(* IEC 61131-3 sources: Elmo_Master/test/Reports_Lasal/C78_20260806_preemption_cleanup_split (part 2) *)

	resourceBusy := FALSE;
	case ResourceKind of
		LMC_OWNER_RESOURCE_LMC_HOME_ENGINE:
			resourceBusy := (OwnershipState[7]$UDINT <> 0) |
				(OwnershipState[8]$UDINT <> 0) |
				(OwnershipState[9]$UDINT <> 0);
		LMC_OWNER_RESOURCE_DS402_HOME_ENGINE:
			resourceBusy := (OwnershipState[10]$UDINT <> 0) |
				(OwnershipState[11]$UDINT <> 0) |
				(OwnershipState[12]$UDINT <> 0);
		LMC_OWNER_RESOURCE_DIAGNOSTICS_SDO_ENGINE:
			resourceBusy := (OwnershipState[13]$UDINT <> 0) |
				(OwnershipState[14]$UDINT <> 0) |
				(OwnershipState[15]$UDINT <> 0);
	else
	end_case;
	if resourceBusy then
		Result := -2;
		RETURN;
	end_if;

	groupLeaseTransition :=
		(OwnerKind = LMC_OWNER_KIND_GROUP) &
		((CommandId = 0x20A4) | (CommandId = 0x7D22) |
		 (CommandId = 0x2048));
	groupStopTransition :=
		(OwnerKind = LMC_OWNER_KIND_GROUP) & (CommandId = 0x2085);

	// A direct safety command against a Group member protects the complete
	// exact lease mask. Unknown Group state widens to the administrative mask
	// and is forced to quarantine after the physical safety observation.
	if (OwnerKind = LMC_OWNER_KIND_DIRECT) & safetyPreemption &
	   (referenceAxisMask <> 0) then
		axisIndex := TO_DINT(Reference);
		recordBase := LMC_OWNER_GLOBAL_SLOTS +
			((axisIndex - 1) * LMC_OWNER_AXIS_STRIDE);
		if (OwnershipState[recordBase + 1] = LMC_OWNER_STATE_GROUP_LEASE) |
		   (OwnershipState[recordBase + 1] = LMC_OWNER_STATE_GROUP_ACTIVE) then
			if (OwnershipState[recordBase + 11]$UDINT <> 0) &
			   (OwnershipState[recordBase + 11]$UDINT <=
			    LMC_OWNER_ROBOT_AXIS_MASK) then
				effectiveAxisMask :=
					OwnershipState[recordBase + 11]$UDINT;
			else
				effectiveAxisMask := LMC_OWNER_ROBOT_AXIS_MASK;
			end_if;
			forceQuarantine := TRUE;
		end_if;
	end_if;

	if groupStopTransition then
		recordBase := LMC_OWNER_GLOBAL_SLOTS;
		if ((OwnershipState[recordBase + 1] = LMC_OWNER_STATE_GROUP_LEASE) |
		    (OwnershipState[recordBase + 1] = LMC_OWNER_STATE_GROUP_ACTIVE)) &
		   (OwnershipState[recordBase + 2] = LMC_OWNER_KIND_GROUP) &
		   (OwnershipState[recordBase + 11]$UDINT =
		    LMC_OWNER_PROFILE_AXIS_MASK) then
			effectiveAxisMask := LMC_OWNER_PROFILE_AXIS_MASK;
		else
			effectiveAxisMask := LMC_OWNER_ROBOT_AXIS_MASK;
			forceQuarantine := TRUE;
		end_if;
	end_if;

	// Repeated safety commands reuse the immutable live lineage. Admission
	// returns +1 for a no-native ACK and +2 for one monotonic PowerOff call.
	repeatCandidate := safetyPreemption &
		((CommandId = LMC_OWNER_COMMAND_AXIS_STOP) |
		 (CommandId = LMC_OWNER_COMMAND_AXIS_POWER) |
		 (CommandId = LMC_OWNER_COMMAND_GROUP_DISABLE) |
		 (CommandId = LMC_OWNER_COMMAND_GROUP_STOP) |
		 (CommandId = LMC_OWNER_COMMAND_GROUP_POWER_OFF));
	if repeatCandidate then
		if OwnerKind = LMC_OWNER_KIND_DIRECT then
			if (Reference >= 1) & (Reference <= LMC_OWNER_AXIS_COUNT) then
			repeatRecordBase := LMC_OWNER_GLOBAL_SLOTS +
				((TO_DINT(Reference) - 1) * LMC_OWNER_AXIS_STRIDE);
			if (OwnershipState[repeatRecordBase + 2] =
			    LMC_OWNER_KIND_DIRECT) &
			   (OwnershipState[repeatRecordBase + 13] =
			    LMC_OWNER_RESOURCE_AXIS) &
			   (OwnershipState[repeatRecordBase + 14] =
			    LMC_OWNER_ADMISSION_SAFETY) then
				repeatFound := TRUE;
			end_if;
			end_if;
		else
			axisIndex := 1;
			while axisIndex <= LMC_OWNER_AXIS_COUNT do
				recordBase := LMC_OWNER_GLOBAL_SLOTS +
					((axisIndex - 1) * LMC_OWNER_AXIS_STRIDE);
				if (OwnershipState[recordBase + 2] =
				    LMC_OWNER_KIND_GROUP) &
				   (OwnershipState[recordBase + 13] =
				    LMC_OWNER_RESOURCE_AXIS) &
				   (OwnershipState[recordBase + 14] =
				    LMC_OWNER_ADMISSION_SAFETY) then
					if repeatFound = FALSE then
						repeatRecordBase := recordBase;
						repeatFound := TRUE;
					elsif (OwnershipState[repeatRecordBase + 4] <>
					       OwnershipState[recordBase + 4]) |
					      (OwnershipState[repeatRecordBase + 5] <>
					       OwnershipState[recordBase + 5]) then
						OwnershipState[24] := 1;
						Result := -3;
						RETURN;
					end_if;
				end_if;
				axisIndex += 1;
			end_while;
		end_if;
	end_if;
	if repeatFound then
		repeatState := OwnershipState[repeatRecordBase + 1];
		if repeatState = LMC_OWNER_STATE_QUARANTINED then
			OwnershipState[24] := 1;
			Result := -3;
			RETURN;
		end_if;
		repeatValid := (repeatState = LMC_OWNER_STATE_RESERVED) |
			(repeatState = LMC_OWNER_STATE_SAFETY_PREEMPTING);
		repeatCommand := OwnershipState[repeatRecordBase + 3];
		repeatReference := OwnershipState[repeatRecordBase + 12];
		repeatOwnerKind := OwnershipState[repeatRecordBase + 2];
		repeatAxisMask := OwnershipState[repeatRecordBase + 11]$UDINT;
		repeatAdmissionToken :=
			OwnershipState[repeatRecordBase + 4]$UDINT;
		repeatOwnerGeneration :=
			OwnershipState[repeatRecordBase + 5]$UDINT;
		repeatSession := OwnershipState[repeatRecordBase + 6]$UDINT;
		repeatSequence := OwnershipState[repeatRecordBase + 7]$UDINT;
		repeatIdentitySize := OwnershipState[repeatRecordBase + 15]$UDINT;
		repeatValid := repeatValid &
			(repeatAxisMask <> 0) &
			(repeatAxisMask <= LMC_OWNER_ROBOT_AXIS_MASK) &
			(repeatAdmissionToken <> 0) &
			(repeatOwnerGeneration <> 0) &
			(repeatSession <> 0) & (repeatSequence <> 0) &
			(((repeatOwnerKind = LMC_OWNER_KIND_DIRECT) &
			  (repeatReference = TO_DINT(Reference)) &
			  ((repeatCommand = LMC_OWNER_COMMAND_AXIS_STOP) |
			   (repeatCommand = LMC_OWNER_COMMAND_AXIS_POWER))) |
			 ((repeatOwnerKind = LMC_OWNER_KIND_GROUP) &
			  (repeatReference = 0x0100) &
			  ((repeatCommand = LMC_OWNER_COMMAND_GROUP_DISABLE) |
			   (repeatCommand = LMC_OWNER_COMMAND_GROUP_STOP) |
			   (repeatCommand = LMC_OWNER_COMMAND_GROUP_POWER_OFF))));
		if repeatValid then
			if repeatState = LMC_OWNER_STATE_RESERVED then
				repeatValidationResult := ValidateAxisOwnershipIdentity(
					CommandId:=repeatCommand$UINT,
					Reference:=repeatReference$UINT,
					ExpectedAxisMask:=repeatAxisMask,
					OwnerKind:=repeatOwnerKind$UINT,
					ResourceKind:=LMC_OWNER_RESOURCE_AXIS,
					AdmissionMode:=LMC_OWNER_ADMISSION_SAFETY,
					CallerSessionEpoch:=repeatSession,
					RequestSequence:=repeatSequence,
					AdmissionToken:=repeatAdmissionToken,
					OwnerGeneration:=repeatOwnerGeneration,
					RequiredPhase:=LMC_OWNER_PHASE_RESERVED,
					pIdentity:=(#OwnershipState[repeatRecordBase + 16])$^void,
					IdentitySize:=repeatIdentitySize);
			else
				repeatValidationResult := ValidateAxisOwnershipIdentity(
				CommandId:=repeatCommand$UINT,
				Reference:=repeatReference$UINT,
				ExpectedAxisMask:=repeatAxisMask,
				OwnerKind:=repeatOwnerKind$UINT,
				ResourceKind:=LMC_OWNER_RESOURCE_AXIS,
				AdmissionMode:=LMC_OWNER_ADMISSION_SAFETY,
				CallerSessionEpoch:=repeatSession,
				RequestSequence:=repeatSequence,
				AdmissionToken:=repeatAdmissionToken,
				OwnerGeneration:=repeatOwnerGeneration,
				RequiredPhase:=LMC_OWNER_PHASE_ACTIVE,
				pIdentity:=(#OwnershipState[repeatRecordBase + 16])$^void,
				IdentitySize:=repeatIdentitySize);
			end_if;
			repeatValid := repeatValidationResult = 0;
		end_if;
		if repeatState = LMC_OWNER_STATE_RESERVED then
			if repeatValid then
				Result := -2;
			else
				OwnershipState[24] := 1;
				Result := -3;
			end_if;
			RETURN;
		end_if;
		if repeatValid then
			axisIndex := 1;
			while axisIndex <= LMC_OWNER_AXIS_COUNT do
				case axisIndex of
					1: axisBit := 0x00000001;
					2: axisBit := 0x00000002;
					3: axisBit := 0x00000004;
					4: axisBit := 0x00000008;
					5: axisBit := 0x00000010;
					6: axisBit := 0x00000020;
					7: axisBit := 0x00000040;
					8: axisBit := 0x00000080;
					9: axisBit := 0x00000100;
				else
					axisBit := 0;
				end_case;
				if (repeatAxisMask and axisBit) <> 0 then
					observerBase := (axisIndex - 1) *
						LMC_OWNER_OBSERVER_STRIDE;
					observerFlags :=
						OwnershipObserverState[observerBase + 5]$UDINT;
					if (OwnershipObserverState[observerBase]$UDINT <>
					    (LMC_OWNER_OBSERVER_MAGIC + TO_UDINT(axisIndex))) |
					   (OwnershipObserverState[observerBase + 1]$UDINT <>
					    repeatAdmissionToken) |
					   (OwnershipObserverState[observerBase + 2]$UDINT <>
					    repeatOwnerGeneration) |
					   ((observerFlags and
					     (0xFFFFFFFF xor LMC_OWNER_OBSERVER_KNOWN_MASK)) <> 0) then
						repeatValid := FALSE;
					end_if;
					if (observerFlags and
					    LMC_OWNER_OBSERVER_PREEMPTED) <> 0 then
						repeatPreemptedSeen := TRUE;
						if (OwnershipObserverState[observerBase + 9] = 0) |
						   (OwnershipObserverState[observerBase + 10] = 0) |
						   (OwnershipObserverState[observerBase + 11] = 0) then
							repeatValid := FALSE;
						end_if;
					elsif (OwnershipObserverState[observerBase + 9] <> 0) |
					      (OwnershipObserverState[observerBase + 10] <> 0) |
					      (OwnershipObserverState[observerBase + 11] <> 0) then
						repeatValid := FALSE;
					end_if;
					if repeatRecordBase = (LMC_OWNER_GLOBAL_SLOTS +
					   ((axisIndex - 1) * LMC_OWNER_AXIS_STRIDE)) then
						repeatEscalated := (observerFlags and
							LMC_OWNER_OBSERVER_POWER_OFF_ESCALATED) <> 0;
						repeatForceQuarantine := (observerFlags and
							LMC_OWNER_OBSERVER_FORCE_QUARANTINE) <> 0;
					else
						if repeatEscalated <>
						   ((observerFlags and
						     LMC_OWNER_OBSERVER_POWER_OFF_ESCALATED) <> 0) then
							repeatValid := FALSE;
						end_if;
						if repeatForceQuarantine <>
						   ((observerFlags and
						     LMC_OWNER_OBSERVER_FORCE_QUARANTINE) <> 0) then
							repeatValid := FALSE;
						end_if;
					end_if;
				end_if;
				axisIndex += 1;
			end_while;
		end_if;
		if repeatValid & (repeatOwnerKind = LMC_OWNER_KIND_DIRECT) then
			if ((repeatAxisMask and referenceAxisMask) <> referenceAxisMask) |
			   ((repeatAxisMask <> referenceAxisMask) &
			    (repeatForceQuarantine = FALSE)) then
				repeatValid := FALSE;
			end_if;
		elsif repeatValid & (repeatOwnerKind = LMC_OWNER_KIND_GROUP) then
			if ((repeatCommand = LMC_OWNER_COMMAND_GROUP_DISABLE) &
			    (repeatAxisMask <> LMC_OWNER_PROFILE_AXIS_MASK)) |
			   ((repeatCommand = LMC_OWNER_COMMAND_GROUP_STOP) &
			    (repeatAxisMask <> LMC_OWNER_PROFILE_AXIS_MASK) &
			    (repeatAxisMask <> LMC_OWNER_ROBOT_AXIS_MASK)) |
			   ((repeatCommand = LMC_OWNER_COMMAND_GROUP_POWER_OFF) &
			    (repeatAxisMask <> LMC_OWNER_ROBOT_AXIS_MASK)) then
				repeatValid := FALSE;
			end_if;
		end_if;
		if repeatValid & repeatEscalated &
		   ((repeatCommand = LMC_OWNER_COMMAND_AXIS_POWER) |
		    (repeatCommand = LMC_OWNER_COMMAND_GROUP_POWER_OFF)) then
			repeatValid := FALSE;
		end_if;
		if repeatValid & repeatRootPresent then
			repeatRootForce :=
				(OwnershipPreemptedIdentityState[
				 LMC_OWNER_PREEMPT_HEADER_BASE + 1]$UDINT and
				 LMC_OWNER_PREEMPT_FLAG_FORCE_QUARANTINE) <> 0;
			if ((OwnershipPreemptedIdentityState[
			     LMC_OWNER_PREEMPT_HEADER_BASE + 1]$UDINT and
			     0x0000FFFF) <> LMC_OWNER_IDENTITY_VERSION) |
			   ((OwnershipPreemptedIdentityState[
			     LMC_OWNER_PREEMPT_HEADER_BASE + 1]$UDINT and
			     0xFFFE0000) <> 0) |
			   (repeatPreemptedSeen = FALSE) then
				repeatValid := FALSE;
			end_if;
			if repeatValid &
			   (repeatRootForce <> repeatForceQuarantine) then
				if repeatRootForce |
				   (repeatForceQuarantine = FALSE) |
				   (repeatEscalated = FALSE) |
				   (repeatOwnerKind <> LMC_OWNER_KIND_GROUP) |
				   (repeatAxisMask <> LMC_OWNER_PROFILE_AXIS_MASK) |
				   ((repeatCommand <> LMC_OWNER_COMMAND_GROUP_DISABLE) &
				    (repeatCommand <> LMC_OWNER_COMMAND_GROUP_STOP)) then
					repeatValid := FALSE;
				end_if;
			end_if;
			axisIndex := 1;
			while axisIndex <= LMC_OWNER_AXIS_COUNT do
				probeRecordBase :=
					(axisIndex - 1) * LMC_OWNER_AXIS_STRIDE;
				if (repeatPreemptedToken = 0) &
				   (OwnershipPreemptedState[probeRecordBase + 1] <>
				    LMC_OWNER_STATE_IDLE) &
				   ((OwnershipPreemptedState[probeRecordBase + 11]$UDINT and
				     repeatAxisMask) <> 0) then
					repeatPreemptedToken := OwnershipPreemptedState[
						probeRecordBase + 4]$UDINT;
					repeatPreemptedGeneration := OwnershipPreemptedState[
						probeRecordBase + 5]$UDINT;
				end_if;
				axisIndex += 1;
			end_while;
			if (repeatPreemptedToken = 0) |
			   (repeatPreemptedGeneration = 0) then
				repeatValid := FALSE;
			end_if;
		elsif repeatValid & repeatPreemptedSeen then
			repeatValid := FALSE;
		end_if;
		if repeatValid then
			if repeatEscalated &
			   (repeatCommand = LMC_OWNER_COMMAND_AXIS_STOP) &
			   ((CommandId = LMC_OWNER_COMMAND_AXIS_STOP) |
			    (CommandId = LMC_OWNER_COMMAND_AXIS_POWER)) then
				repeatMode := 1;
			elsif repeatEscalated &
			      ((repeatCommand = LMC_OWNER_COMMAND_GROUP_STOP) |
			       (repeatCommand = LMC_OWNER_COMMAND_GROUP_DISABLE)) &
			      ((CommandId = LMC_OWNER_COMMAND_GROUP_STOP) |
			       (CommandId = LMC_OWNER_COMMAND_GROUP_DISABLE) |
			       (CommandId = LMC_OWNER_COMMAND_GROUP_POWER_OFF)) then
				repeatMode := 1;
			elsif repeatCommand = TO_DINT(CommandId) then
				if (repeatCommand = LMC_OWNER_COMMAND_AXIS_STOP) |
				   (repeatCommand = LMC_OWNER_COMMAND_GROUP_STOP) then
					identityCompareResult := _memcmp(
						ptr1:=pIdentity,
						ptr2:=#OwnershipState[repeatRecordBase + 16],
						cntr:=repeatIdentitySize);
					if identityCompareResult = 0 then
						repeatMode := 1;
					end_if;
				else
					repeatMode := 1;
				end_if;
			elsif (repeatCommand = LMC_OWNER_COMMAND_AXIS_POWER) &
			      (CommandId = LMC_OWNER_COMMAND_AXIS_STOP) then
				repeatMode := 1;
			elsif (repeatCommand = LMC_OWNER_COMMAND_GROUP_POWER_OFF) &
			      ((CommandId = LMC_OWNER_COMMAND_GROUP_STOP) |
			       (CommandId = LMC_OWNER_COMMAND_GROUP_DISABLE)) then
				repeatMode := 1;
			elsif (repeatCommand = LMC_OWNER_COMMAND_AXIS_STOP) &
			      (CommandId = LMC_OWNER_COMMAND_AXIS_POWER) then
				if repeatEscalated then
					repeatMode := 1;
				else
					repeatMode := 2;
				end_if;
			elsif ((repeatCommand = LMC_OWNER_COMMAND_GROUP_STOP) |
			       (repeatCommand = LMC_OWNER_COMMAND_GROUP_DISABLE)) &
			      (CommandId = LMC_OWNER_COMMAND_GROUP_POWER_OFF) then
				if repeatEscalated then
					repeatMode := 1;
				else
					repeatMode := 2;
				end_if;
			end_if;
		end_if;
		if repeatValid = FALSE then
			OwnershipState[24] := 1;
			Result := -3;
			RETURN;
		end_if;
	end_if;
	if repeatRootPresent & safetyPreemption & (repeatMode = 0) then
		Result := -2;
		RETURN;
	end_if;

	if repeatMode = 0 then
	axisIndex := 1;
	while axisIndex <= LMC_OWNER_AXIS_COUNT do
		case axisIndex of
			1: axisBit := 0x00000001;
			2: axisBit := 0x00000002;
			3: axisBit := 0x00000004;
			4: axisBit := 0x00000008;
			5: axisBit := 0x00000010;
			6: axisBit := 0x00000020;
			7: axisBit := 0x00000040;
			8: axisBit := 0x00000080;
			9: axisBit := 0x00000100;
		else
			axisBit := 0;
		end_case;
		if (effectiveAxisMask and axisBit) <> 0 then
			recordBase := LMC_OWNER_GLOBAL_SLOTS +
				((axisIndex - 1) * LMC_OWNER_AXIS_STRIDE);
			if (OwnershipState[recordBase] <> axisIndex) |
			   (OwnershipState[recordBase + 35]$UDINT <>
			    (LMC_OWNER_AXIS_RECORD_MAGIC + TO_UDINT(axisIndex))) then
				Result := -3;
				RETURN;
			end_if;
			existingState := OwnershipState[recordBase + 1];
			existingOwnerKind := OwnershipState[recordBase + 2];
			if (existingState = LMC_OWNER_STATE_IDLE) &
			   ((OwnershipState[recordBase + 2] <> 0) |
			    (OwnershipState[recordBase + 3] <> 0) |
			    (OwnershipState[recordBase + 4] <> 0) |
			    (OwnershipState[recordBase + 5] <> 0) |
			    (OwnershipState[recordBase + 6] <> 0) |
			    (OwnershipState[recordBase + 7] <> 0) |
			    (OwnershipState[recordBase + 11] <> 0) |
			    (OwnershipState[recordBase + 13] <> 0) |
			    (OwnershipState[recordBase + 14] <> 0) |
			    (OwnershipState[recordBase + 15] <> 0)) then
				Result := -3;
				RETURN;
			end_if;
			if safetyPreemption &
			   (existingState = LMC_OWNER_STATE_SAFETY_PREEMPTING) then
				Result := -2;
				RETURN;
			end_if;

			// Validate the complete current identity header before it can be
			// copied to a lease or preemption bank.
			existingIdentityValid := existingState = LMC_OWNER_STATE_IDLE;
			if existingState <> LMC_OWNER_STATE_IDLE then
				if (OwnershipState[recordBase + 15] < 0) |
				   (OwnershipState[recordBase + 15]$UDINT > 1320) then
					Result := -3;
					RETURN;
				end_if;
				if existingOwnerKind = LMC_OWNER_KIND_GROUP then
					identityHeaderBase := LMC_OWNER_IDENTITY_GROUP_HEADER_BASE;
					existingIdentityValid :=
						(OwnershipIdentityState[identityHeaderBase]$UDINT =
						 LMC_OWNER_IDENTITY_GROUP_MAGIC) &
						(OwnershipIdentityState[identityHeaderBase + 1] =
						 LMC_OWNER_IDENTITY_VERSION) &
						(OwnershipIdentityState[identityHeaderBase + 2]$UDINT =
						 OwnershipState[recordBase + 15]$UDINT) &
						(OwnershipIdentityState[identityHeaderBase + 3]$UDINT =
						 OwnershipState[recordBase + 4]$UDINT) &
						(OwnershipIdentityState[identityHeaderBase + 4]$UDINT =
						 OwnershipState[recordBase + 5]$UDINT) &
						(OwnershipIdentityState[identityHeaderBase + 5]$UDINT =
						 OwnershipState[recordBase + 11]$UDINT) &
						(OwnershipIdentityState[identityHeaderBase + 6]$UDINT =
						 OwnershipState[recordBase + 6]$UDINT) &
						(OwnershipIdentityState[identityHeaderBase + 7]$UDINT =
						 OwnershipState[recordBase + 7]$UDINT) &
						(OwnershipIdentityState[identityHeaderBase + 8]$UDINT =
						 (TO_UDINT(OwnershipState[recordBase + 3]) or
						  (TO_UDINT(OwnershipState[recordBase + 12]) shl 16))) &
						(OwnershipIdentityState[identityHeaderBase + 9]$UDINT =
						 (TO_UDINT(OwnershipState[recordBase + 2]) or
						  (TO_UDINT(OwnershipState[recordBase + 13]) shl 8) or
						  (TO_UDINT(OwnershipState[recordBase + 14]) shl 16)));
				else
					identityHeaderBase := LMC_OWNER_IDENTITY_AXIS_HEADER_BASE +
						((axisIndex - 1) *
						 LMC_OWNER_IDENTITY_AXIS_HEADER_STRIDE);
					identityTailSize := 0;
					if OwnershipState[recordBase + 15]$UDINT >
					   LMC_OWNER_IDENTITY_PREFIX_BYTES then
						identityTailSize :=
							OwnershipState[recordBase + 15]$UDINT -
							LMC_OWNER_IDENTITY_PREFIX_BYTES;
					end_if;
					if (OwnershipState[recordBase + 12] < 1) |
					   (OwnershipState[recordBase + 12] >
					    LMC_OWNER_AXIS_COUNT) |
					   (identityTailSize > 8) then
						Result := -3;
						RETURN;
					end_if;
					identityTailOffset :=
						TO_UDINT(OwnershipState[recordBase + 12] - 1) * 8;
					existingIdentityValid :=
						(OwnershipIdentityState[identityHeaderBase]$UDINT =
						 (LMC_OWNER_IDENTITY_AXIS_MAGIC + TO_UDINT(axisIndex))) &
						(OwnershipIdentityState[identityHeaderBase + 1] =
						 LMC_OWNER_IDENTITY_VERSION) &
						(OwnershipIdentityState[identityHeaderBase + 2]$UDINT =
						 OwnershipState[recordBase + 15]$UDINT) &
						(OwnershipIdentityState[identityHeaderBase + 3]$UDINT =
						 OwnershipState[recordBase + 4]$UDINT) &
						(OwnershipIdentityState[identityHeaderBase + 4]$UDINT =
						 OwnershipState[recordBase + 5]$UDINT) &
						(OwnershipIdentityState[identityHeaderBase + 5]$UDINT =
						 OwnershipState[recordBase + 11]$UDINT) &
						(OwnershipIdentityState[identityHeaderBase + 6]$UDINT =
						 OwnershipState[recordBase + 6]$UDINT) &
						(OwnershipIdentityState[identityHeaderBase + 7]$UDINT =
						 OwnershipState[recordBase + 7]$UDINT) &
						(OwnershipIdentityState[identityHeaderBase + 8]$UDINT =
						 (TO_UDINT(OwnershipState[recordBase + 3]) or
						  (TO_UDINT(OwnershipState[recordBase + 12]) shl 16))) &
						(OwnershipIdentityState[identityHeaderBase + 9]$UDINT =
						 (TO_UDINT(OwnershipState[recordBase + 2]) or
						  (TO_UDINT(OwnershipState[recordBase + 13]) shl 8) or
						  (TO_UDINT(OwnershipState[recordBase + 14]) shl 16))) &
						(OwnershipIdentityState[identityHeaderBase + 10]$UDINT =
						 identityTailOffset) &
						(OwnershipIdentityState[identityHeaderBase + 11]$UDINT =
						 identityTailSize);
				end_if;
				if existingIdentityValid = FALSE then
					Result := -3;
					RETURN;
				end_if;
				// Every member of one captured tuple was created from one request.
				// Prove complete membership and byte-exact prefix coherence before
				// any backup publication or live ownership mutation.
				existingIdentityPrefixSize :=
					OwnershipState[recordBase + 15]$UDINT;
				if existingIdentityPrefixSize >
				   LMC_OWNER_IDENTITY_PREFIX_BYTES then
					existingIdentityPrefixSize :=
						LMC_OWNER_IDENTITY_PREFIX_BYTES;
				end_if;
				if (OwnershipState[recordBase + 4]$UDINT = 0) |
				   (OwnershipState[recordBase + 5]$UDINT = 0) |
				   (OwnershipState[recordBase + 6]$UDINT = 0) |
				   (OwnershipState[recordBase + 7]$UDINT = 0) |
				   (OwnershipState[recordBase + 11]$UDINT = 0) |
				   (OwnershipState[recordBase + 11]$UDINT >
				    LMC_OWNER_ROBOT_AXIS_MASK) |
				   ((OwnershipState[recordBase + 11]$UDINT and axisBit) = 0) then
					Result := -3;
					RETURN;
				end_if;
				probeAxisIndex := 1;
				while probeAxisIndex <= LMC_OWNER_AXIS_COUNT do
					case probeAxisIndex of
						1: probeAxisBit := 0x00000001;
						2: probeAxisBit := 0x00000002;
						3: probeAxisBit := 0x00000004;
						4: probeAxisBit := 0x00000008;
						5: probeAxisBit := 0x00000010;
						6: probeAxisBit := 0x00000020;
						7: probeAxisBit := 0x00000040;
						8: probeAxisBit := 0x00000080;
						9: probeAxisBit := 0x00000100;
					else
						probeAxisBit := 0;
					end_case;
					probeRecordBase := LMC_OWNER_GLOBAL_SLOTS +
						((probeAxisIndex - 1) * LMC_OWNER_AXIS_STRIDE);
					if (OwnershipState[recordBase + 11]$UDINT and
					    probeAxisBit) <> 0 then
						if (OwnershipState[probeRecordBase] <>
						    probeAxisIndex) |
						   (OwnershipState[probeRecordBase + 35]$UDINT <>
						    (LMC_OWNER_AXIS_RECORD_MAGIC +
						     TO_UDINT(probeAxisIndex))) |
						   (OwnershipState[probeRecordBase + 1] <>
						    OwnershipState[recordBase + 1]) |
						   (OwnershipState[probeRecordBase + 2] <>
						    OwnershipState[recordBase + 2]) |
						   (OwnershipState[probeRecordBase + 3] <>
						    OwnershipState[recordBase + 3]) |
						   (OwnershipState[probeRecordBase + 4]$UDINT <>
						    OwnershipState[recordBase + 4]$UDINT) |
						   (OwnershipState[probeRecordBase + 5]$UDINT <>
						    OwnershipState[recordBase + 5]$UDINT) |
						   (OwnershipState[probeRecordBase + 6]$UDINT <>
						    OwnershipState[recordBase + 6]$UDINT) |
						   (OwnershipState[probeRecordBase + 7]$UDINT <>
						    OwnershipState[recordBase + 7]$UDINT) |
						   (OwnershipState[probeRecordBase + 11]$UDINT <>
						    OwnershipState[recordBase + 11]$UDINT) |
						   (OwnershipState[probeRecordBase + 12] <>
						    OwnershipState[recordBase + 12]) |
						   (OwnershipState[probeRecordBase + 13] <>
						    OwnershipState[recordBase + 13]) |
						   (OwnershipState[probeRecordBase + 14] <>
						    OwnershipState[recordBase + 14]) |
						   (OwnershipState[probeRecordBase + 15]$UDINT <>
						    OwnershipState[recordBase + 15]$UDINT) then
							Result := -3;
							RETURN;
						end_if;
						identityCompareResult := _memcmp(
							ptr1:=#OwnershipState[recordBase + 16],
							ptr2:=#OwnershipState[probeRecordBase + 16],
							cntr:=existingIdentityPrefixSize);
						if identityCompareResult <> 0 then
							Result := -3;
							RETURN;
						end_if;
					elsif (OwnershipState[probeRecordBase + 4]$UDINT =
					       OwnershipState[recordBase + 4]$UDINT) |
					      (OwnershipState[probeRecordBase + 5]$UDINT =
					       OwnershipState[recordBase + 5]$UDINT) then
						Result := -3;
						RETURN;
					end_if;
					probeAxisIndex += 1;
				end_while;
			end_if;

			if existingOwnerKind = LMC_OWNER_KIND_GROUP then
				preemptedGroupOwner :=
					preemptedGroupOwner or
					(existingState <> LMC_OWNER_STATE_IDLE);
				if existingState = LMC_OWNER_STATE_GROUP_ACTIVE then
					existingGroupActive := TRUE;
				end_if;
			end_if;
			if safetyPreemption &
			   (existingState <> LMC_OWNER_STATE_IDLE) then
				preemptCapture := TRUE;
			end_if;
			if safetyPreemption &
			   ((existingOwnerKind = LMC_OWNER_KIND_LMC_HOME) |
			    (existingOwnerKind = LMC_OWNER_KIND_DS402_HOME) |
			    (existingOwnerKind = LMC_OWNER_KIND_ENCODER)) then
				cleanupRequiredMask := cleanupRequiredMask or axisBit;
				case OwnershipState[recordBase + 13] of
					LMC_OWNER_RESOURCE_LMC_HOME_ENGINE:
						existingIdentityValid :=
							(OwnershipState[7]$UDINT =
							 OwnershipState[recordBase + 4]$UDINT) &
							(OwnershipState[8]$UDINT =
							 OwnershipState[recordBase + 5]$UDINT) &
							(OwnershipState[9]$UDINT =
							 OwnershipState[recordBase + 11]$UDINT);
					LMC_OWNER_RESOURCE_DS402_HOME_ENGINE:
						existingIdentityValid :=
							(OwnershipState[10]$UDINT =
							 OwnershipState[recordBase + 4]$UDINT) &
							(OwnershipState[11]$UDINT =
							 OwnershipState[recordBase + 5]$UDINT) &
							(OwnershipState[12]$UDINT =
							 OwnershipState[recordBase + 11]$UDINT);
					LMC_OWNER_RESOURCE_DIAGNOSTICS_SDO_ENGINE:
						existingIdentityValid :=
							(OwnershipState[13]$UDINT =
							 OwnershipState[recordBase + 4]$UDINT) &
							(OwnershipState[14]$UDINT =
							 OwnershipState[recordBase + 5]$UDINT) &
							(OwnershipState[15]$UDINT =
							 OwnershipState[recordBase + 11]$UDINT);
				else
					existingIdentityValid := FALSE;
				end_case;
				if existingIdentityValid = FALSE then
					Result := -3;
					RETURN;
				end_if;
			end_if;

			if groupLeaseTransition then
				if (OwnershipState[recordBase + 1] <>
				    LMC_OWNER_STATE_GROUP_LEASE) |
				   (OwnershipState[recordBase + 2] <>
				    LMC_OWNER_KIND_GROUP) |
				   (OwnershipState[recordBase + 11]$UDINT <>
				    effectiveAxisMask) |
				   (OwnershipState[recordBase + 12] <> TO_DINT(Reference)) |
				   (OwnershipState[recordBase + 6]$UDINT <>
				    CallerSessionEpoch) |
				   (OwnershipState[recordBase + 4]$UDINT = 0) |
				   (OwnershipState[recordBase + 5]$UDINT = 0) then
					Result := -2;
					RETURN;
				end_if;
				if selectedFound = FALSE then
					existingToken := OwnershipState[recordBase + 4]$UDINT;
					existingGeneration :=
						OwnershipState[recordBase + 5]$UDINT;
					selectedFound := TRUE;
				elsif (existingToken <>
				       OwnershipState[recordBase + 4]$UDINT) |
				      (existingGeneration <>
				       OwnershipState[recordBase + 5]$UDINT) then
					Result := -3;
					RETURN;
				end_if;
				leaseCapture := TRUE;
			elsif groupStopTransition & (forceQuarantine = FALSE) then
				if ((OwnershipState[recordBase + 1] <>
				     LMC_OWNER_STATE_GROUP_LEASE) &
				    (OwnershipState[recordBase + 1] <>
				     LMC_OWNER_STATE_GROUP_ACTIVE)) |
				   (OwnershipState[recordBase + 2] <>
				    LMC_OWNER_KIND_GROUP) |
				   (OwnershipState[recordBase + 11]$UDINT <>
				    effectiveAxisMask) |
				   (OwnershipState[recordBase + 12] <> TO_DINT(Reference)) |
				   (OwnershipState[recordBase + 4]$UDINT = 0) |
				   (OwnershipState[recordBase + 5]$UDINT = 0) then
					Result := -2;
					RETURN;
				end_if;
				if selectedFound = FALSE then
					existingToken := OwnershipState[recordBase + 4]$UDINT;
					existingGeneration :=
						OwnershipState[recordBase + 5]$UDINT;
					selectedFound := TRUE;
				elsif (existingToken <>
				       OwnershipState[recordBase + 4]$UDINT) |
				      (existingGeneration <>
				       OwnershipState[recordBase + 5]$UDINT) then
					Result := -3;
					RETURN;
				end_if;
				if existingState = LMC_OWNER_STATE_GROUP_LEASE then
					leaseCapture := TRUE;
				end_if;
			elsif safetyPreemption then
				if OwnershipState[recordBase + 1] =
				   LMC_OWNER_STATE_QUARANTINED then
					forceQuarantine := TRUE;
				end_if;
				if (existingOwnerKind = LMC_OWNER_KIND_GROUP) &
				   (existingState = LMC_OWNER_STATE_GROUP_LEASE) then
					leaseCapture := TRUE;
				end_if;
			else
				if OwnershipState[recordBase + 1] <>
				   LMC_OWNER_STATE_IDLE then
					Result := -2;
					RETURN;
				elsif (OwnershipState[recordBase + 4]$UDINT <> 0) |
				      (OwnershipState[recordBase + 5]$UDINT <> 0) |
				      (OwnershipState[recordBase + 11]$UDINT <> 0) |
				      (OwnershipState[recordBase + 13] <> 0) then
					Result := -3;
					RETURN;
				end_if;
			end_if;
			if leaseCapture &
			   (existingState = LMC_OWNER_STATE_GROUP_LEASE) then
				observersIdle := TRUE;
				observerBase := (axisIndex - 1) *
					LMC_OWNER_OBSERVER_STRIDE;
				observerIndex := 0;
				while observerIndex < LMC_OWNER_OBSERVER_STRIDE do
					if OwnershipObserverState[
					   observerBase + observerIndex] <> 0 then
						observersIdle := FALSE;
					end_if;
					observerIndex += 1;
				end_while;
				if observersIdle = FALSE then
					Result := -3;
					RETURN;
				end_if;
			end_if;
		end_if;
		axisIndex += 1;
	end_while;
	end_if;

	if leaseCapture & leaseAvailable then
		Result := -3;
		RETURN;
	end_if;
	if leaseAvailable then
		existingIdentityValid :=
			(OwnershipLeaseIdentityState[
			 LMC_OWNER_LEASE_IDENTITY_HEADER_BASE]$UDINT =
			 LMC_OWNER_LEASE_IDENTITY_MAGIC) &
			(OwnershipLeaseIdentityState[
			 LMC_OWNER_LEASE_IDENTITY_HEADER_BASE + 1] =
			 LMC_OWNER_IDENTITY_VERSION) &
			(OwnershipLeaseIdentityState[
			 LMC_OWNER_LEASE_IDENTITY_HEADER_BASE + 2]$UDINT = 1) &
			(OwnershipLeaseIdentityState[
			 LMC_OWNER_LEASE_IDENTITY_HEADER_BASE + 3]$UDINT <> 0) &
			(OwnershipLeaseIdentityState[
			 LMC_OWNER_LEASE_IDENTITY_HEADER_BASE + 4]$UDINT <> 0) &
			(OwnershipLeaseIdentityState[
			 LMC_OWNER_LEASE_IDENTITY_HEADER_BASE + 5]$UDINT =
			 LMC_OWNER_PROFILE_AXIS_MASK) &
			(OwnershipLeaseIdentityState[
			 LMC_OWNER_LEASE_IDENTITY_HEADER_BASE + 6]$UDINT <> 0) &
			(OwnershipLeaseIdentityState[
			 LMC_OWNER_LEASE_IDENTITY_HEADER_BASE + 7]$UDINT <> 0) &
			(OwnershipLeaseIdentityState[
			 LMC_OWNER_LEASE_IDENTITY_HEADER_BASE + 8]$UDINT =
			 (TO_UDINT(0x2047) or (TO_UDINT(0x0100) shl 16))) &
			(OwnershipLeaseIdentityState[
			 LMC_OWNER_LEASE_IDENTITY_HEADER_BASE + 9]$UDINT =
			 (TO_UDINT(LMC_OWNER_KIND_GROUP) or
			  (TO_UDINT(LMC_OWNER_RESOURCE_AXIS) shl 8) or
			  (TO_UDINT(LMC_OWNER_ADMISSION_ORDINARY) shl 16)));
		leaseFirstRecordBase := -1;
		axisIndex := 1;
		while axisIndex <= LMC_OWNER_AXIS_COUNT do
			case axisIndex of
				1: axisBit := 0x00000001;
				2: axisBit := 0x00000002;
				3: axisBit := 0x00000004;
				4: axisBit := 0x00000008;
				5: axisBit := 0x00000010;
				6: axisBit := 0x00000020;
				7: axisBit := 0x00000040;
				8: axisBit := 0x00000080;
				9: axisBit := 0x00000100;
			else
				axisBit := 0;
			end_case;
			recordBase := (axisIndex - 1) * LMC_OWNER_AXIS_STRIDE;
			if (OwnershipLeaseState[recordBase] <> axisIndex) |
			   (OwnershipLeaseState[recordBase + 35]$UDINT <>
			    (LMC_OWNER_AXIS_RECORD_MAGIC + TO_UDINT(axisIndex))) then
				existingIdentityValid := FALSE;
			end_if;
			if (OwnershipLeaseIdentityState[
			    LMC_OWNER_LEASE_IDENTITY_HEADER_BASE + 5]$UDINT and
			    axisBit) <> 0 then
				if (OwnershipLeaseState[recordBase + 1] <>
				    LMC_OWNER_STATE_GROUP_LEASE) |
				   (OwnershipLeaseState[recordBase + 2] <>
				    LMC_OWNER_KIND_GROUP) |
				   (OwnershipLeaseState[recordBase + 3] <> 0x2047) |
				   (OwnershipLeaseState[recordBase + 4]$UDINT <>
				    OwnershipLeaseIdentityState[
				     LMC_OWNER_LEASE_IDENTITY_HEADER_BASE + 3]$UDINT) |
				   (OwnershipLeaseState[recordBase + 5]$UDINT <>
				    OwnershipLeaseIdentityState[
				     LMC_OWNER_LEASE_IDENTITY_HEADER_BASE + 4]$UDINT) |
				   (OwnershipLeaseState[recordBase + 6]$UDINT <>
				    OwnershipLeaseIdentityState[
				     LMC_OWNER_LEASE_IDENTITY_HEADER_BASE + 6]$UDINT) |
				   (OwnershipLeaseState[recordBase + 7]$UDINT <>
				    OwnershipLeaseIdentityState[
				     LMC_OWNER_LEASE_IDENTITY_HEADER_BASE + 7]$UDINT) |
				   (OwnershipLeaseState[recordBase + 11]$UDINT <>
				    LMC_OWNER_PROFILE_AXIS_MASK) |
				   (OwnershipLeaseState[recordBase + 12] <> 0x0100) |
				   (OwnershipLeaseState[recordBase + 13] <>
				    LMC_OWNER_RESOURCE_AXIS) |
				   (OwnershipLeaseState[recordBase + 14] <>
				    LMC_OWNER_ADMISSION_ORDINARY) |
				   (OwnershipLeaseState[recordBase + 15]$UDINT <> 1) |
				   (OwnershipLeaseState[recordBase + 16]$UDINT <> 1) then
					existingIdentityValid := FALSE;
				end_if;
				identityIndex := 17;
				while identityIndex <= 31 do
					if OwnershipLeaseState[recordBase + identityIndex] <> 0 then
						existingIdentityValid := FALSE;
					end_if;
					identityIndex += 1;
				end_while;
				if leaseFirstRecordBase < 0 then
					leaseFirstRecordBase := recordBase;
				else
					identityCompareResult := _memcmp(
						ptr1:=#OwnershipLeaseState[leaseFirstRecordBase + 16],
						ptr2:=#OwnershipLeaseState[recordBase + 16], cntr:=1);
					if identityCompareResult <> 0 then
						existingIdentityValid := FALSE;
					end_if;
				end_if;
			else
				if (OwnershipLeaseState[recordBase + 4]$UDINT =
				    OwnershipLeaseIdentityState[
				     LMC_OWNER_LEASE_IDENTITY_HEADER_BASE + 3]$UDINT) |
				   (OwnershipLeaseState[recordBase + 5]$UDINT =
				    OwnershipLeaseIdentityState[
				     LMC_OWNER_LEASE_IDENTITY_HEADER_BASE + 4]$UDINT) then
					existingIdentityValid := FALSE;
				end_if;
				identityIndex := 1;
				while identityIndex <= 34 do
					if OwnershipLeaseState[recordBase + identityIndex] <> 0 then
						existingIdentityValid := FALSE;
					end_if;
					identityIndex += 1;
				end_while;
			end_if;
			axisIndex += 1;
		end_while;
		identityIndex := 0;
		while identityIndex < LMC_OWNER_IDENTITY_SUFFIX_DINTS do
			if OwnershipLeaseIdentityState[identityIndex] <> 0 then
				existingIdentityValid := FALSE;
			end_if;
			identityIndex += 1;
		end_while;
		if (existingIdentityValid = FALSE) | (leaseFirstRecordBase < 0) then
			Result := -3;
			RETURN;
		end_if;
	end_if;
	if existingGroupActive & groupStopTransition &
	   (leaseAvailable = FALSE) then
		forceQuarantine := TRUE;
	end_if;
	if repeatMode > 0 then
		if repeatRootPresent then
			repeatPreemptCopyResult := CopyAxisOwnershipPreemption(
				PreemptedAdmissionToken:=repeatPreemptedToken,
				PreemptedOwnerGeneration:=repeatPreemptedGeneration,
				pDest:=#repeatPreemptProbe[0], DestSize:=144);
			if repeatPreemptCopyResult <> -4 then
				OwnershipState[24] := 1;
				Result := -3;
				RETURN;
			end_if;
		end_if;
		pEffectiveAxisMask^ := repeatAxisMask;
		pAdmissionToken^ := repeatAdmissionToken;
		pOwnerGeneration^ := repeatOwnerGeneration;
		Result := repeatMode;
		RETURN;
	end_if;

	nextToken := OwnershipState[1]$UDINT + 1;
	if nextToken = 0 then
		nextToken := 1;
	end_if;
	if (groupLeaseTransition | groupStopTransition) &
	   (forceQuarantine = FALSE) & (existingGeneration <> 0) then
		nextGeneration := existingGeneration;
	else
		nextGeneration := OwnershipState[2]$UDINT + 1;
		if nextGeneration = 0 then
			nextGeneration := 1;
		end_if;
	end_if;

	// Publish exact backup banks only after every validation has passed.
	if leaseCapture then
		OwnershipLeaseIdentityState[
			LMC_OWNER_LEASE_IDENTITY_HEADER_BASE] := 0;
		_memset(dest:=#OwnershipLeaseState[0], usByte:=0,
			cntr:=sizeof(OwnershipLeaseState));
		_memset(dest:=#OwnershipLeaseIdentityState[0], usByte:=0,
			cntr:=sizeof(OwnershipLeaseIdentityState));
		_memcpy(ptr1:=#OwnershipLeaseState[0],
			ptr2:=#OwnershipState[LMC_OWNER_GLOBAL_SLOTS],
			cntr:=sizeof(OwnershipLeaseState));
		_memcpy(ptr1:=#OwnershipLeaseIdentityState[0],
			ptr2:=#OwnershipIdentityState[0],
			cntr:=LMC_OWNER_IDENTITY_SUFFIX_BYTES);
		identityIndex := 1;
		while identityIndex <= 9 do
			OwnershipLeaseIdentityState[
				LMC_OWNER_LEASE_IDENTITY_HEADER_BASE + identityIndex] :=
				OwnershipIdentityState[
				 LMC_OWNER_IDENTITY_GROUP_HEADER_BASE + identityIndex];
			identityIndex += 1;
		end_while;
		OwnershipLeaseIdentityState[
			LMC_OWNER_LEASE_IDENTITY_HEADER_BASE]$UDINT :=
			LMC_OWNER_LEASE_IDENTITY_MAGIC;
		leaseAvailable := TRUE;
	end_if;

	if preemptCapture then
		OwnershipPreemptedIdentityState[
			LMC_OWNER_PREEMPT_HEADER_BASE] := 0;
		_memset(dest:=#OwnershipPreemptedState[0], usByte:=0,
			cntr:=sizeof(OwnershipPreemptedState));
		_memset(dest:=#OwnershipPreemptedIdentityState[0], usByte:=0,
			cntr:=sizeof(OwnershipPreemptedIdentityState));
		_memcpy(ptr1:=#OwnershipPreemptedState[0],
			ptr2:=#OwnershipState[LMC_OWNER_GLOBAL_SLOTS],
			cntr:=sizeof(OwnershipPreemptedState));
		_memcpy(ptr1:=#OwnershipPreemptedIdentityState[0],
			ptr2:=#OwnershipIdentityState[0],
			cntr:=LMC_OWNER_IDENTITY_SUFFIX_BYTES);
		_memcpy(ptr1:=#OwnershipPreemptedIdentityState[
			LMC_OWNER_PREEMPT_OBSERVER_BASE],
			ptr2:=#OwnershipObserverState[0],
			cntr:=sizeof(OwnershipObserverState));
		OwnershipPreemptedIdentityState[
			LMC_OWNER_PREEMPT_HEADER_BASE + 1]$UDINT :=
			LMC_OWNER_IDENTITY_VERSION;
		if forceQuarantine then
			OwnershipPreemptedIdentityState[
				LMC_OWNER_PREEMPT_HEADER_BASE + 1]$UDINT :=
				OwnershipPreemptedIdentityState[
				 LMC_OWNER_PREEMPT_HEADER_BASE + 1]$UDINT or
				LMC_OWNER_PREEMPT_FLAG_FORCE_QUARANTINE;
		end_if;
		OwnershipPreemptedIdentityState[
			LMC_OWNER_PREEMPT_HEADER_BASE + 2]$UDINT := nextToken;
		OwnershipPreemptedIdentityState[
			LMC_OWNER_PREEMPT_HEADER_BASE + 3]$UDINT := nextGeneration;
		OwnershipPreemptedIdentityState[
			LMC_OWNER_PREEMPT_HEADER_BASE + 4]$UDINT := effectiveAxisMask;
		OwnershipPreemptedIdentityState[
			LMC_OWNER_PREEMPT_HEADER_BASE + 5]$UDINT := CallerSessionEpoch;
		OwnershipPreemptedIdentityState[
			LMC_OWNER_PREEMPT_HEADER_BASE + 6]$UDINT := RequestSequence;
		OwnershipPreemptedIdentityState[
			LMC_OWNER_PREEMPT_HEADER_BASE + 7]$UDINT :=
			identityPackedCommand;
		OwnershipPreemptedIdentityState[
			LMC_OWNER_PREEMPT_HEADER_BASE + 8]$UDINT := cleanupRequiredMask;
		OwnershipPreemptedIdentityState[
			LMC_OWNER_PREEMPT_HEADER_BASE + 9] := 0;
		OwnershipPreemptedIdentityState[
			LMC_OWNER_PREEMPT_HEADER_BASE]$UDINT :=
			LMC_OWNER_PREEMPT_IDENTITY_MAGIC;
	end_if;

	OwnershipState[1]$UDINT := nextToken;
	if nextGeneration > OwnershipState[2]$UDINT then
		OwnershipState[2]$UDINT := nextGeneration;
	end_if;

	identityPrefixSize := IdentitySize;
	if identityPrefixSize > LMC_OWNER_IDENTITY_PREFIX_BYTES then
		identityPrefixSize := LMC_OWNER_IDENTITY_PREFIX_BYTES;
	end_if;
	identityTailSize := 0;
	if IdentitySize > LMC_OWNER_IDENTITY_PREFIX_BYTES then
		identityTailSize := IdentitySize - LMC_OWNER_IDENTITY_PREFIX_BYTES;
	end_if;
	identityTailOffset := 0;
	if OwnerKind <> LMC_OWNER_KIND_GROUP then
		identityTailOffset := TO_UDINT(Reference - 1) * 8;
	end_if;
	axisIndex := 1;
	while axisIndex <= LMC_OWNER_AXIS_COUNT do
		case axisIndex of
			1: axisBit := 0x00000001;
			2: axisBit := 0x00000002;
			3: axisBit := 0x00000004;
			4: axisBit := 0x00000008;
			5: axisBit := 0x00000010;
			6: axisBit := 0x00000020;
			7: axisBit := 0x00000040;
			8: axisBit := 0x00000080;
			9: axisBit := 0x00000100;
		else
			axisBit := 0;
		end_case;
		if (effectiveAxisMask and axisBit) <> 0 then
			identityHeaderBase := LMC_OWNER_IDENTITY_AXIS_HEADER_BASE +
				((axisIndex - 1) *
				 LMC_OWNER_IDENTITY_AXIS_HEADER_STRIDE);
			OwnershipIdentityState[identityHeaderBase] := 0;
		end_if;
		axisIndex += 1;
	end_while;
	if (OwnerKind = LMC_OWNER_KIND_GROUP) | preemptedGroupOwner then
		OwnershipIdentityState[
			LMC_OWNER_IDENTITY_GROUP_HEADER_BASE] := 0;
		if safetyPreemption = FALSE then
			_memset(dest:=#OwnershipIdentityState[0], usByte:=0,
				cntr:=LMC_OWNER_IDENTITY_SUFFIX_BYTES);
		end_if;
		identityIndex := 0;
		while identityIndex < 10 do
			OwnershipIdentityState[
				LMC_OWNER_IDENTITY_GROUP_HEADER_BASE + identityIndex] := 0;
			identityIndex += 1;
		end_while;
	end_if;
	if (OwnerKind <> LMC_OWNER_KIND_GROUP) & (identityTailSize > 0) then
		_memset(dest:=#OwnershipIdentityState[
			TO_DINT(identityTailOffset / 4)], usByte:=0,
			cntr:=identityTailSize);
	end_if;
	if identityTailSize > 0 then
		_memcpy(ptr1:=#OwnershipIdentityState[
			TO_DINT(identityTailOffset / 4)],
			ptr2:=pIdentityBytes + LMC_OWNER_IDENTITY_PREFIX_BYTES,
			cntr:=identityTailSize);
	end_if;

	axisIndex := 1;
	while axisIndex <= LMC_OWNER_AXIS_COUNT do
		case axisIndex of
			1: axisBit := 0x00000001;
			2: axisBit := 0x00000002;
			3: axisBit := 0x00000004;
			4: axisBit := 0x00000008;
			5: axisBit := 0x00000010;
			6: axisBit := 0x00000020;
			7: axisBit := 0x00000040;
			8: axisBit := 0x00000080;
			9: axisBit := 0x00000100;
		else
			axisBit := 0;
		end_case;
		if (effectiveAxisMask and axisBit) <> 0 then
			recordBase := LMC_OWNER_GLOBAL_SLOTS +
				((axisIndex - 1) * LMC_OWNER_AXIS_STRIDE);
			observerBase := (axisIndex - 1) * LMC_OWNER_OBSERVER_STRIDE;
			existingState := OwnershipState[recordBase + 1];
			existingOwnerKind := OwnershipState[recordBase + 2];
			observerFlags := 0;
			if (CommandId = 0x2047) | (CommandId = 0x20A4) |
			   (CommandId = 0x7D22) | (CommandId = 0x2085) then
				observerFlags := observerFlags or
					LMC_OWNER_OBSERVER_RETURN_GROUP_LEASE;
			end_if;
			if groupLeaseTransition | groupStopTransition then
				observerFlags := observerFlags or
					LMC_OWNER_OBSERVER_RESTORE_GROUP_LEASE;
			end_if;
			if safetyPreemption & (existingState <> LMC_OWNER_STATE_IDLE) then
				observerFlags := observerFlags or
					LMC_OWNER_OBSERVER_PREEMPTED;
			end_if;
			if existingState = LMC_OWNER_STATE_GROUP_ACTIVE then
				observerFlags := observerFlags or
					LMC_OWNER_OBSERVER_GROUP_ACTIVE_PREEMPTED;
			end_if;
			if (existingOwnerKind = LMC_OWNER_KIND_LMC_HOME) |
			   (existingOwnerKind = LMC_OWNER_KIND_DS402_HOME) |
			   (existingOwnerKind = LMC_OWNER_KIND_ENCODER) then
				observerFlags := observerFlags or
					LMC_OWNER_OBSERVER_PREEMPTED_SPECIAL;
			end_if;
			if existingState = LMC_OWNER_STATE_QUARANTINED then
				observerFlags := observerFlags or
					LMC_OWNER_OBSERVER_FORCE_QUARANTINE;
			end_if;
			if forceQuarantine then
				observerFlags := observerFlags or
					LMC_OWNER_OBSERVER_FORCE_QUARANTINE;
			end_if;
			observerIndex := 0;
			while observerIndex < LMC_OWNER_OBSERVER_STRIDE do
				OwnershipObserverState[observerBase + observerIndex] := 0;
				observerIndex += 1;
			end_while;
			OwnershipObserverState[observerBase]$UDINT :=
				LMC_OWNER_OBSERVER_MAGIC + TO_UDINT(axisIndex);
			OwnershipObserverState[observerBase + 5]$UDINT := observerFlags;
			OwnershipObserverState[observerBase + 9]$UDINT :=
				OwnershipState[recordBase + 4]$UDINT;
			OwnershipObserverState[observerBase + 10]$UDINT :=
				OwnershipState[recordBase + 5]$UDINT;
			OwnershipObserverState[observerBase + 11] := existingState;
			OwnershipState[recordBase] := axisIndex;
			OwnershipState[recordBase + 1] := LMC_OWNER_STATE_RESERVED;
			OwnershipState[recordBase + 2] := TO_DINT(OwnerKind);
			OwnershipState[recordBase + 3] := TO_DINT(CommandId);
			OwnershipState[recordBase + 4]$UDINT := nextToken;
			OwnershipState[recordBase + 5]$UDINT := nextGeneration;
			OwnershipState[recordBase + 6]$UDINT := CallerSessionEpoch;
			OwnershipState[recordBase + 7]$UDINT := RequestSequence;
			OwnershipState[recordBase + 8]$UDINT := ops.tAbsolute;
			OwnershipState[recordBase + 9]$UDINT := ops.tAbsolute;
			OwnershipState[recordBase + 10] := 0;
			OwnershipState[recordBase + 11]$UDINT := effectiveAxisMask;
			OwnershipState[recordBase + 12] := TO_DINT(Reference);
			OwnershipState[recordBase + 13] := TO_DINT(ResourceKind);
			OwnershipState[recordBase + 14] := TO_DINT(AdmissionMode);
			OwnershipState[recordBase + 15] := TO_DINT(IdentitySize);
			_memset(dest:=#OwnershipState[recordBase + 16], usByte:=0,
				cntr:=LMC_OWNER_IDENTITY_PREFIX_BYTES);
			if identityPrefixSize > 0 then
				_memcpy(ptr1:=#OwnershipState[recordBase + 16],
					ptr2:=pIdentityBytes, cntr:=identityPrefixSize);
			end_if;
			OwnershipState[recordBase + 32] := 0;
			OwnershipState[recordBase + 33] := 0;
			OwnershipState[recordBase + 34] := 0;
			OwnershipState[recordBase + 35]$UDINT :=
				LMC_OWNER_AXIS_RECORD_MAGIC + TO_UDINT(axisIndex);

			identityHeaderBase := LMC_OWNER_IDENTITY_AXIS_HEADER_BASE +
				((axisIndex - 1) *
				 LMC_OWNER_IDENTITY_AXIS_HEADER_STRIDE);
			_memset(dest:=#OwnershipIdentityState[identityHeaderBase],
				usByte:=0,
				cntr:=LMC_OWNER_IDENTITY_AXIS_HEADER_STRIDE * 4);
			if OwnerKind <> LMC_OWNER_KIND_GROUP then
				OwnershipIdentityState[identityHeaderBase + 1] :=
					LMC_OWNER_IDENTITY_VERSION;
				OwnershipIdentityState[identityHeaderBase + 2]$UDINT :=
					IdentitySize;
				OwnershipIdentityState[identityHeaderBase + 3]$UDINT :=
					nextToken;
				OwnershipIdentityState[identityHeaderBase + 4]$UDINT :=
					nextGeneration;
				OwnershipIdentityState[identityHeaderBase + 5]$UDINT :=
					effectiveAxisMask;
				OwnershipIdentityState[identityHeaderBase + 6]$UDINT :=
					CallerSessionEpoch;
				OwnershipIdentityState[identityHeaderBase + 7]$UDINT :=
					RequestSequence;
				OwnershipIdentityState[identityHeaderBase + 8]$UDINT :=
					identityPackedCommand;
				OwnershipIdentityState[identityHeaderBase + 9]$UDINT :=
					identityPackedOwner;
				OwnershipIdentityState[identityHeaderBase + 10]$UDINT :=
					identityTailOffset;
				OwnershipIdentityState[identityHeaderBase + 11]$UDINT :=
					identityTailSize;
				OwnershipIdentityState[identityHeaderBase]$UDINT :=
					LMC_OWNER_IDENTITY_AXIS_MAGIC + TO_UDINT(axisIndex);
			end_if;
		end_if;
		axisIndex += 1;
	end_while;
	if OwnerKind = LMC_OWNER_KIND_GROUP then
		identityHeaderBase := LMC_OWNER_IDENTITY_GROUP_HEADER_BASE;
		OwnershipIdentityState[identityHeaderBase + 1] :=
			LMC_OWNER_IDENTITY_VERSION;
		OwnershipIdentityState[identityHeaderBase + 2]$UDINT := IdentitySize;
		OwnershipIdentityState[identityHeaderBase + 3]$UDINT := nextToken;
		OwnershipIdentityState[identityHeaderBase + 4]$UDINT := nextGeneration;
		OwnershipIdentityState[identityHeaderBase + 5]$UDINT :=
			effectiveAxisMask;
		OwnershipIdentityState[identityHeaderBase + 6]$UDINT :=
			CallerSessionEpoch;
		OwnershipIdentityState[identityHeaderBase + 7]$UDINT :=
			RequestSequence;
		OwnershipIdentityState[identityHeaderBase + 8]$UDINT :=
			identityPackedCommand;
		OwnershipIdentityState[identityHeaderBase + 9]$UDINT :=
			identityPackedOwner;
		OwnershipIdentityState[identityHeaderBase]$UDINT :=
			LMC_OWNER_IDENTITY_GROUP_MAGIC;
	end_if;

	case ResourceKind of
		LMC_OWNER_RESOURCE_LMC_HOME_ENGINE:
			OwnershipState[7]$UDINT := nextToken;
			OwnershipState[8]$UDINT := nextGeneration;
			OwnershipState[9]$UDINT := effectiveAxisMask;
		LMC_OWNER_RESOURCE_DS402_HOME_ENGINE:
			OwnershipState[10]$UDINT := nextToken;
			OwnershipState[11]$UDINT := nextGeneration;
			OwnershipState[12]$UDINT := effectiveAxisMask;
		LMC_OWNER_RESOURCE_DIAGNOSTICS_SDO_ENGINE:
			OwnershipState[13]$UDINT := nextToken;
			OwnershipState[14]$UDINT := nextGeneration;
			OwnershipState[15]$UDINT := effectiveAxisMask;
	else
	end_case;

	pEffectiveAxisMask^ := effectiveAxisMask;
	pAdmissionToken^ := nextToken;
	pOwnerGeneration^ := nextGeneration;
	Result := 0;

END_FUNCTION

FUNCTION GLOBAL LMCControlCommandService::ValidateAxisOwnership
	VAR_INPUT
		CommandId 	: UINT;
		Reference 	: UINT;
		ExpectedAxisMask 	: UDINT;
		OwnerKind 	: UINT;
		ResourceKind 	: UINT;
		AdmissionMode 	: UINT;
		CallerSessionEpoch 	: UDINT;
		RequestSequence 	: UDINT;
		AdmissionToken 	: UDINT;
		OwnerGeneration 	: UDINT;
		RequiredPhase 	: UINT;
	END_VAR
	VAR_OUTPUT
		Result 	: DINT;
	END_VAR
	VAR
		axisIndex : DINT;
		axisBit : UDINT;
		referenceAxisMask : UDINT;
		recordBase : DINT;
		expectedState : DINT;
		resourceValid : BOOL;
		tupleValid : BOOL;
	END_VAR

	Result := -1;
	if (ExpectedAxisMask = 0) |
	   (ExpectedAxisMask > LMC_OWNER_ROBOT_AXIS_MASK) |
	   (AdmissionToken = 0) | (OwnerGeneration = 0) |
	   (CallerSessionEpoch = 0) | (RequestSequence = 0) |
	   ((RequiredPhase <> LMC_OWNER_PHASE_RESERVED) &
	    (RequiredPhase <> LMC_OWNER_PHASE_ACTIVE) &
	    (RequiredPhase <> LMC_OWNER_PHASE_SESSION_CLOSED_ROLLBACK)) then
		RETURN;
	end_if;
	referenceAxisMask := 0;
	case Reference of
		1: referenceAxisMask := 0x00000001;
		2: referenceAxisMask := 0x00000002;
		3: referenceAxisMask := 0x00000004;
		4: referenceAxisMask := 0x00000008;
		5: referenceAxisMask := 0x00000010;
		6: referenceAxisMask := 0x00000020;
		7: referenceAxisMask := 0x00000040;
		8: referenceAxisMask := 0x00000080;
		9: referenceAxisMask := 0x00000100;
	else
	end_case;
	tupleValid := FALSE;
	case CommandId of
		0x2022:
			tupleValid :=
				(OwnerKind = LMC_OWNER_KIND_DIRECT) &
				(ResourceKind = LMC_OWNER_RESOURCE_AXIS) &
				(AdmissionMode = LMC_OWNER_ADMISSION_SAFETY) &
				(referenceAxisMask <> 0) &
				(ExpectedAxisMask <= LMC_OWNER_ROBOT_AXIS_MASK) &
				((ExpectedAxisMask and referenceAxisMask) <> 0);
		0x2023:
			tupleValid :=
				(OwnerKind = LMC_OWNER_KIND_DIRECT) &
				(ResourceKind = LMC_OWNER_RESOURCE_AXIS) &
				(referenceAxisMask <> 0) &
				(((AdmissionMode = LMC_OWNER_ADMISSION_ORDINARY) &
				  (ExpectedAxisMask = referenceAxisMask)) |
				 ((AdmissionMode = LMC_OWNER_ADMISSION_SAFETY) &
				  (ExpectedAxisMask <= LMC_OWNER_ROBOT_AXIS_MASK) &
				  ((ExpectedAxisMask and referenceAxisMask) <> 0)));
		0x2024, 0x209F, 0x20A0, 0x20A2:
			tupleValid :=
				(OwnerKind = LMC_OWNER_KIND_DIRECT) &
				(ResourceKind = LMC_OWNER_RESOURCE_AXIS) &
				(AdmissionMode = LMC_OWNER_ADMISSION_ORDINARY) &
				(referenceAxisMask <> 0) &
				(ExpectedAxisMask = referenceAxisMask);
		0x2047, 0x20A4, 0x7D22:
			tupleValid :=
				(OwnerKind = LMC_OWNER_KIND_GROUP) &
				(ResourceKind = LMC_OWNER_RESOURCE_AXIS) &
				(AdmissionMode = LMC_OWNER_ADMISSION_ORDINARY) &
				(Reference = 0x0100) &
				(ExpectedAxisMask = LMC_OWNER_PROFILE_AXIS_MASK);
		0x2048:
			tupleValid :=
				(OwnerKind = LMC_OWNER_KIND_GROUP) &
				(ResourceKind = LMC_OWNER_RESOURCE_AXIS) &
				(AdmissionMode = LMC_OWNER_ADMISSION_SAFETY) &
				(Reference = 0x0100) &
				(ExpectedAxisMask = LMC_OWNER_PROFILE_AXIS_MASK);
		0x2085:
			tupleValid :=
				(OwnerKind = LMC_OWNER_KIND_GROUP) &
				(ResourceKind = LMC_OWNER_RESOURCE_AXIS) &
				(AdmissionMode = LMC_OWNER_ADMISSION_SAFETY) &
				(Reference = 0x0100) &
				((ExpectedAxisMask = LMC_OWNER_PROFILE_AXIS_MASK) |
				 (ExpectedAxisMask = LMC_OWNER_ROBOT_AXIS_MASK));
		0x2049, 0x204A:
			tupleValid :=
				(OwnerKind = LMC_OWNER_KIND_GROUP) &
				(ResourceKind = LMC_OWNER_RESOURCE_AXIS) &
				(AdmissionMode = LMC_OWNER_ADMISSION_ORDINARY) &
				(Reference = 0x0100) &
				(ExpectedAxisMask = LMC_OWNER_ROBOT_AXIS_MASK);
		0x204B:
			tupleValid :=
				(OwnerKind = LMC_OWNER_KIND_GROUP) &
				(ResourceKind = LMC_OWNER_RESOURCE_AXIS) &
				(AdmissionMode = LMC_OWNER_ADMISSION_SAFETY) &
				(Reference = 0x0100) &
				(ExpectedAxisMask = LMC_OWNER_ROBOT_AXIS_MASK);
		0x20E7:
			tupleValid :=
				(OwnerKind = LMC_OWNER_KIND_GROUP) &
				(ResourceKind = LMC_OWNER_RESOURCE_AXIS) &
				(AdmissionMode = LMC_OWNER_ADMISSION_LIFECYCLE) &
				(Reference = 0x0100) &
				(ExpectedAxisMask = LMC_OWNER_ROBOT_AXIS_MASK);
		0x7D13:
			tupleValid :=
				(OwnerKind = LMC_OWNER_KIND_LMC_HOME) &
				(ResourceKind = LMC_OWNER_RESOURCE_LMC_HOME_ENGINE) &
				(AdmissionMode = LMC_OWNER_ADMISSION_LIFECYCLE) &
				(referenceAxisMask <> 0) &
				(referenceAxisMask <= 0x00000008) &
				(ExpectedAxisMask = referenceAxisMask);
		0x7D15:
			tupleValid :=
				(OwnerKind = LMC_OWNER_KIND_DS402_HOME) &
				(ResourceKind = LMC_OWNER_RESOURCE_DS402_HOME_ENGINE) &
				(AdmissionMode = LMC_OWNER_ADMISSION_LIFECYCLE) &
				(referenceAxisMask <> 0) &
				(referenceAxisMask <= 0x00000008) &
				(ExpectedAxisMask = referenceAxisMask);
		0x7E53:
			tupleValid :=
				(OwnerKind = LMC_OWNER_KIND_ENCODER) &
				(ResourceKind = LMC_OWNER_RESOURCE_DIAGNOSTICS_SDO_ENGINE) &
				(AdmissionMode = LMC_OWNER_ADMISSION_LIFECYCLE) &
				(referenceAxisMask <> 0) &
				(referenceAxisMask <= 0x00000008) &
				(ExpectedAxisMask = referenceAxisMask);
	else
	end_case;
	if tupleValid = FALSE then
		RETURN;
	end_if;
	expectedState := LMC_OWNER_STATE_RESERVED;
	if RequiredPhase = LMC_OWNER_PHASE_SESSION_CLOSED_ROLLBACK then
		if (CommandId <> 0x7D15) |
		   (OwnerKind <> LMC_OWNER_KIND_DS402_HOME) |
		   (ResourceKind <> LMC_OWNER_RESOURCE_DS402_HOME_ENGINE) |
		   (AdmissionMode <> LMC_OWNER_ADMISSION_LIFECYCLE) then
			RETURN;
		end_if;
		expectedState := LMC_OWNER_STATE_QUARANTINED;
	elsif RequiredPhase = LMC_OWNER_PHASE_ACTIVE then
		if AdmissionMode = LMC_OWNER_ADMISSION_SAFETY then
			if (OwnerKind = LMC_OWNER_KIND_DIRECT) |
			   (OwnerKind = LMC_OWNER_KIND_GROUP) then
				expectedState := LMC_OWNER_STATE_SAFETY_PREEMPTING;
			else
				RETURN;
			end_if;
		else
			case OwnerKind of
				LMC_OWNER_KIND_DIRECT:
					expectedState := LMC_OWNER_STATE_DIRECT_ACTIVE;
				LMC_OWNER_KIND_GROUP:
					expectedState := LMC_OWNER_STATE_GROUP_ACTIVE;
				LMC_OWNER_KIND_LMC_HOME:
					expectedState := LMC_OWNER_STATE_LMC_HOME_ACTIVE;
				LMC_OWNER_KIND_DS402_HOME:
					expectedState := LMC_OWNER_STATE_DS402_HOME_ACTIVE;
				LMC_OWNER_KIND_ENCODER:
					expectedState := LMC_OWNER_STATE_TW20_QUEUED;
			else
				RETURN;
			end_case;
		end_if;
	end_if;
	if (OwnershipState[0]$UDINT <> LMC_OWNER_TABLE_MAGIC) |
	   (OwnershipState[3]$UDINT = 0) |
	   (OwnershipState[24] <> 0) then
		Result := -3;
		RETURN;
	end_if;

	resourceValid :=
		(ResourceKind = LMC_OWNER_RESOURCE_AXIS) &
		(OwnershipState[7]$UDINT <> AdmissionToken) &
		(OwnershipState[8]$UDINT <> OwnerGeneration) &
		(OwnershipState[10]$UDINT <> AdmissionToken) &
		(OwnershipState[11]$UDINT <> OwnerGeneration) &
		(OwnershipState[13]$UDINT <> AdmissionToken) &
		(OwnershipState[14]$UDINT <> OwnerGeneration);
	case ResourceKind of
		LMC_OWNER_RESOURCE_LMC_HOME_ENGINE:
			resourceValid :=
				(OwnershipState[7]$UDINT = AdmissionToken) &
				(OwnershipState[8]$UDINT = OwnerGeneration) &
				(OwnershipState[9]$UDINT = ExpectedAxisMask);
		LMC_OWNER_RESOURCE_DS402_HOME_ENGINE:
			resourceValid :=
				(OwnershipState[10]$UDINT = AdmissionToken) &
				(OwnershipState[11]$UDINT = OwnerGeneration) &
				(OwnershipState[12]$UDINT = ExpectedAxisMask);
		LMC_OWNER_RESOURCE_DIAGNOSTICS_SDO_ENGINE:
			resourceValid :=
				(OwnershipState[13]$UDINT = AdmissionToken) &
				(OwnershipState[14]$UDINT = OwnerGeneration) &
				(OwnershipState[15]$UDINT = ExpectedAxisMask);
	else
	end_case;
	if resourceValid = FALSE then
		Result := -2;
		RETURN;
	end_if;

	axisIndex := 1;
	while axisIndex <= LMC_OWNER_AXIS_COUNT do
		case axisIndex of
			1: axisBit := 0x00000001;
			2: axisBit := 0x00000002;
			3: axisBit := 0x00000004;
			4: axisBit := 0x00000008;
			5: axisBit := 0x00000010;
			6: axisBit := 0x00000020;
			7: axisBit := 0x00000040;
			8: axisBit := 0x00000080;
			9: axisBit := 0x00000100;
		else
			axisBit := 0;
		end_case;
		recordBase := LMC_OWNER_GLOBAL_SLOTS +
			((axisIndex - 1) * LMC_OWNER_AXIS_STRIDE);
		if (ExpectedAxisMask and axisBit) <> 0 then
			if (OwnershipState[recordBase + 1] =
			    LMC_OWNER_STATE_QUARANTINED) &
			   (RequiredPhase <>
			    LMC_OWNER_PHASE_SESSION_CLOSED_ROLLBACK) then
				Result := -3;
				RETURN;
			elsif (OwnershipState[recordBase] <> axisIndex) |
			      (OwnershipState[recordBase + 35]$UDINT <>
			       (LMC_OWNER_AXIS_RECORD_MAGIC + TO_UDINT(axisIndex))) |
			      (OwnershipState[recordBase + 1] <> expectedState) |
			      (OwnershipState[recordBase + 2] <> TO_DINT(OwnerKind)) |
			      (OwnershipState[recordBase + 3] <> TO_DINT(CommandId)) |
			      (OwnershipState[recordBase + 4]$UDINT <> AdmissionToken) |
			      (OwnershipState[recordBase + 5]$UDINT <> OwnerGeneration) |
			      (OwnershipState[recordBase + 6]$UDINT <>
			       CallerSessionEpoch) |
			      (OwnershipState[recordBase + 7]$UDINT <> RequestSequence) |
			      (OwnershipState[recordBase + 11]$UDINT <>
			       ExpectedAxisMask) |
			      (OwnershipState[recordBase + 12] <> TO_DINT(Reference)) |
			      (OwnershipState[recordBase + 13] <>
			       TO_DINT(ResourceKind)) |
			      (OwnershipState[recordBase + 14] <>
			       TO_DINT(AdmissionMode)) then
				Result := -2;
				RETURN;
			end_if;
		elsif (OwnershipState[recordBase + 4]$UDINT = AdmissionToken) |
		      (OwnershipState[recordBase + 5]$UDINT = OwnerGeneration) then
			Result := -2;
			RETURN;
		end_if;
		axisIndex += 1;
	end_while;

	Result := 0;

END_FUNCTION

FUNCTION GLOBAL LMCControlCommandService::CommitAxisOwnership
	VAR_INPUT
		CommandId : UINT;
		Reference : UINT;
		ExpectedAxisMask : UDINT;
		CallerSessionEpoch : UDINT;
		RequestSequence : UDINT;
		AdmissionToken : UDINT;
		OwnerGeneration : UDINT;
	END_VAR
	VAR_OUTPUT
		Result : DINT;
	END_VAR
	VAR
		axisIndex : DINT;
		axisBit : UDINT;
		probeAxisBit : UDINT;
		recordBase : DINT;
		observerBase : DINT;
		ownerKind : UINT;
		resourceKind : UINT;
		admissionMode : UINT;
		activeState : DINT;
		observerFlags : UDINT;
		rebaseUpdateResult : DINT;
	END_VAR

	Result := -1;
	if (ExpectedAxisMask = 0) |
	   (ExpectedAxisMask > LMC_OWNER_ROBOT_AXIS_MASK) then
		RETURN;
	end_if;
	// Read the lease kind from one selected axis without changing any record.
	axisIndex := 1;
	while axisIndex <= LMC_OWNER_AXIS_COUNT do
		case axisIndex of
			1: axisBit := 0x00000001;
			2: axisBit := 0x00000002;
			3: axisBit := 0x00000004;
			4: axisBit := 0x00000008;
			5: axisBit := 0x00000010;
			6: axisBit := 0x00000020;
			7: axisBit := 0x00000040;
			8: axisBit := 0x00000080;
			9: axisBit := 0x00000100;
		else
			axisBit := 0;
		end_case;
		if (ExpectedAxisMask and axisBit) <> 0 then
			recordBase := LMC_OWNER_GLOBAL_SLOTS +
				((axisIndex - 1) * LMC_OWNER_AXIS_STRIDE);
			ownerKind := OwnershipState[recordBase + 2]$UINT;
			resourceKind := OwnershipState[recordBase + 13]$UINT;
			admissionMode := OwnershipState[recordBase + 14]$UINT;
			exit;
		end_if;
		axisIndex += 1;
	end_while;
	if axisIndex > LMC_OWNER_AXIS_COUNT then
		RETURN;
	end_if;

	// Validate the complete mask exactly once before the first mutation.
	Result := ValidateAxisOwnership(
		CommandId:=CommandId,
		Reference:=Reference,
		ExpectedAxisMask:=ExpectedAxisMask,
		OwnerKind:=ownerKind,
		ResourceKind:=resourceKind,
		AdmissionMode:=admissionMode,
		CallerSessionEpoch:=CallerSessionEpoch,
		RequestSequence:=RequestSequence,
		AdmissionToken:=AdmissionToken,
		OwnerGeneration:=OwnerGeneration,
		RequiredPhase:=LMC_OWNER_PHASE_RESERVED);
	if Result <> 0 then
		RETURN;
	end_if;
	// Arm before the first owner mutation and before Diagnostics can call the
	// SDO executor. A later pre-dispatch failure intentionally still requires
	// Home because false-positive coordinate recovery is safer than a gap.
	if LMC_AXIS_REBASE_BARRIER_ENABLED &
	   (CommandId = 0x7E53) &
	   (ownerKind = LMC_OWNER_KIND_ENCODER) &
	   (resourceKind = LMC_OWNER_RESOURCE_DIAGNOSTICS_SDO_ENGINE) &
	   (admissionMode = LMC_OWNER_ADMISSION_LIFECYCLE) &
	   (Reference >= 1) & (Reference <= 4) &
	   (ExpectedAxisMask = axisBit) &
	   (OwnershipState[recordBase + 15]$UDINT = 72) &
	   (OwnershipState[recordBase + 25]$UINT = 2) &
	   (OwnershipState[recordBase + 26]$UINT = Reference) &
	   (OwnershipState[recordBase + 27]$UDINT = 1) then
		rebaseUpdateResult := UpdateAxisRebaseRequiredState(
			SetAxisMask:=ExpectedAxisMask, ClearAxisMask:=0);
		if rebaseUpdateResult <> 0 then
			Result := rebaseUpdateResult;
			RETURN;
		end_if;
	end_if;
	if admissionMode = LMC_OWNER_ADMISSION_SAFETY then
		activeState := LMC_OWNER_STATE_SAFETY_PREEMPTING;
	else
		case ownerKind of
			LMC_OWNER_KIND_GROUP:
				activeState := LMC_OWNER_STATE_GROUP_ACTIVE;
			LMC_OWNER_KIND_LMC_HOME:
				activeState := LMC_OWNER_STATE_LMC_HOME_ACTIVE;
			LMC_OWNER_KIND_DS402_HOME:
				activeState := LMC_OWNER_STATE_DS402_HOME_ACTIVE;
			LMC_OWNER_KIND_ENCODER:
				activeState := LMC_OWNER_STATE_TW20_QUEUED;
		else
			activeState := LMC_OWNER_STATE_DIRECT_ACTIVE;
		end_case;
	end_if;

	axisIndex := 1;
	while axisIndex <= LMC_OWNER_AXIS_COUNT do
		case axisIndex of
			1: axisBit := 0x00000001;
			2: axisBit := 0x00000002;
			3: axisBit := 0x00000004;
			4: axisBit := 0x00000008;
			5: axisBit := 0x00000010;
			6: axisBit := 0x00000020;
			7: axisBit := 0x00000040;
			8: axisBit := 0x00000080;
			9: axisBit := 0x00000100;
		else
			axisBit := 0;
		end_case;
		if (ExpectedAxisMask and axisBit) <> 0 then
			recordBase := LMC_OWNER_GLOBAL_SLOTS +
				((axisIndex - 1) * LMC_OWNER_AXIS_STRIDE);
			observerBase := (axisIndex - 1) * LMC_OWNER_OBSERVER_STRIDE;
			observerFlags :=
				OwnershipObserverState[observerBase + 5]$UDINT;
			OwnershipState[recordBase + 1] := activeState;
			OwnershipState[recordBase + 9]$UDINT := ops.tAbsolute;
			OwnershipState[recordBase + 10] := 0;
			OwnershipObserverState[observerBase]$UDINT :=
				LMC_OWNER_OBSERVER_MAGIC + TO_UDINT(axisIndex);
			OwnershipObserverState[observerBase + 1]$UDINT := AdmissionToken;
			OwnershipObserverState[observerBase + 2]$UDINT := OwnerGeneration;
			OwnershipObserverState[observerBase + 3] := 0;
			OwnershipObserverState[observerBase + 4] := 0;
			OwnershipObserverState[observerBase + 5]$UDINT := observerFlags;
			OwnershipObserverState[observerBase + 6] := 0;
			OwnershipObserverState[observerBase + 7] := 0;
			OwnershipObserverState[observerBase + 8] := 0;
		end_if;
		axisIndex += 1;
	end_while;
	Result := 0;

END_FUNCTION

FUNCTION GLOBAL LMCControlCommandService::RollbackAxisOwnership
	VAR_INPUT
		AdmissionToken : UDINT;
		OwnerGeneration : UDINT;
		CallerSessionEpoch : UDINT;
		RequestSequence : UDINT;
		Reason : DINT;
	END_VAR
	VAR_OUTPUT
		Result : DINT;
	END_VAR
	VAR
		axisIndex : DINT;
		axisBit : UDINT;
		probeAxisIndex : DINT;
		probeAxisBit : UDINT;
		recordBase : DINT;
		probeRecordBase : DINT;
		firstRecordBase : DINT;
		observerBase : DINT;
		observerIndex : DINT;
		identityIndex : DINT;
		clearIndex : DINT;
		expectedAxisMask : UDINT;
		expectedResourceKind : DINT;
		expectedReference : DINT;
		expectedCommandId : DINT;
		expectedOwnerKind : DINT;
		expectedAdmissionMode : DINT;
		expectedSession : UDINT;
		expectedSequence : UDINT;
		expectedIdentitySize : UDINT;
		observerFlags : UDINT;
		preemptedToken : UDINT;
		preemptedGeneration : UDINT;
		snapshotToken : UDINT;
		snapshotGeneration : UDINT;
		snapshotSession : UDINT;
		snapshotSequence : UDINT;
		snapshotMask : UDINT;
		snapshotCommand : DINT;
		snapshotReference : DINT;
		snapshotOwnerKind : DINT;
		snapshotResourceKind : DINT;
		snapshotAdmissionMode : DINT;
		snapshotState : DINT;
		snapshotIdentitySize : UDINT;
		leaseExpectedMask : UDINT;
		restoredGroupMask : UDINT;
		restoredGroupToken : UDINT;
		restoredGroupGeneration : UDINT;
		restoredGroupSession : UDINT;
		restoredGroupSequence : UDINT;
		restoredGroupIdentitySize : UDINT;
		restoredGroupCommand : DINT;
		restoredGroupReference : DINT;
		restoredGroupState : DINT;
		restoredGroupAdmissionMode : DINT;
		preemptFlags : UDINT;
		cleanupRequiredMask : UDINT;
		cleanupCompleteMask : UDINT;
		identityHeaderBase : DINT;
		identityCompareResult : UDINT;
		identitySize : UDINT;
		identityExpectedSize : UDINT;
		identityPrefixSize : UDINT;
		identityTailSize : UDINT;
		identityTailOffset : UDINT;
		identityPackedCommand : UDINT;
		identityPackedOwner : UDINT;
		matched : BOOL;
		resourceValid : BOOL;
		restorePreempt : BOOL;
		restoreLease : BOOL;
		preemptBankValid : BOOL;
		leaseBankValid : BOOL;
		identityShapeValid : BOOL;
		snapshotTupleValid : BOOL;
		observerSnapshotValid : BOOL;
		observersIdle : BOOL;
		restoredGroupActive : BOOL;
		restoredGroupFound : BOOL;
		restoredNonSafetyFound : BOOL;
		groupHeaderPublished : BOOL;
	END_VAR

	Result := -1;
	if (AdmissionToken = 0) | (OwnerGeneration = 0) |
	   (CallerSessionEpoch = 0) | (RequestSequence = 0) then
		RETURN;
	end_if;
	matched := FALSE;
	restorePreempt := FALSE;
	restoreLease := FALSE;
	expectedAxisMask := 0;
	expectedResourceKind := 0;
	expectedReference := 0;
	expectedCommandId := 0;
	expectedOwnerKind := 0;
	expectedAdmissionMode := 0;
	expectedSession := 0;
	expectedSequence := 0;
	expectedIdentitySize := 0;
	firstRecordBase := -1;
	restoredGroupActive := FALSE;
	restoredGroupFound := FALSE;
	restoredNonSafetyFound := FALSE;
	// Derive one immutable complete set before validating or changing any member.
	axisIndex := 1;
	while axisIndex <= LMC_OWNER_AXIS_COUNT do
		recordBase := LMC_OWNER_GLOBAL_SLOTS +
			((axisIndex - 1) * LMC_OWNER_AXIS_STRIDE);
		if (OwnershipState[recordBase + 4]$UDINT = AdmissionToken) &
		   (OwnershipState[recordBase + 5]$UDINT = OwnerGeneration) then
			matched := TRUE;
			if expectedAxisMask = 0 then
				expectedAxisMask := OwnershipState[recordBase + 11]$UDINT;
				expectedResourceKind := OwnershipState[recordBase + 13];
				expectedReference := OwnershipState[recordBase + 12];
				expectedCommandId := OwnershipState[recordBase + 3];
				expectedOwnerKind := OwnershipState[recordBase + 2];
				expectedAdmissionMode := OwnershipState[recordBase + 14];
				expectedSession := OwnershipState[recordBase + 6]$UDINT;
				expectedSequence := OwnershipState[recordBase + 7]$UDINT;
				expectedIdentitySize := OwnershipState[recordBase + 15]$UDINT;
				firstRecordBase := recordBase;
			elsif (expectedAxisMask <>
			       OwnershipState[recordBase + 11]$UDINT) |
			      (expectedResourceKind <>
			       OwnershipState[recordBase + 13]) |
			      (expectedReference <>
			       OwnershipState[recordBase + 12]) |
			      (expectedCommandId <>
			       OwnershipState[recordBase + 3]) |
			      (expectedOwnerKind <>
			       OwnershipState[recordBase + 2]) |
			      (expectedAdmissionMode <>
			       OwnershipState[recordBase + 14]) |
			      (expectedSession <>
			       OwnershipState[recordBase + 6]$UDINT) |
			      (expectedSequence <>
			       OwnershipState[recordBase + 7]$UDINT) |
			      (expectedIdentitySize <>
			       OwnershipState[recordBase + 15]$UDINT) then
				Result := -2;
				RETURN;
			end_if;
		end_if;
		axisIndex += 1;
	end_while;
	if matched = FALSE then
		Result := -2;
		RETURN;
	end_if;
	if (expectedAxisMask = 0) |
	   (expectedAxisMask > LMC_OWNER_ROBOT_AXIS_MASK) then
		Result := -2;
		RETURN;
	end_if;

	// Validate every expected member and reject every extra matching member.
	axisIndex := 1;
	while axisIndex <= LMC_OWNER_AXIS_COUNT do
		case axisIndex of
			1: axisBit := 0x00000001;
			2: axisBit := 0x00000002;
			3: axisBit := 0x00000004;
			4: axisBit := 0x00000008;
			5: axisBit := 0x00000010;
			6: axisBit := 0x00000020;
			7: axisBit := 0x00000040;
			8: axisBit := 0x00000080;
			9: axisBit := 0x00000100;
		else
			axisBit := 0;
		end_case;
		recordBase := LMC_OWNER_GLOBAL_SLOTS +
			((axisIndex - 1) * LMC_OWNER_AXIS_STRIDE);
		if (expectedAxisMask and axisBit) <> 0 then
			if (OwnershipState[recordBase] <> axisIndex) |
			   (OwnershipState[recordBase + 35]$UDINT <>
			    (LMC_OWNER_AXIS_RECORD_MAGIC + TO_UDINT(axisIndex))) |
			   (OwnershipState[recordBase + 4]$UDINT <> AdmissionToken) |
			   (OwnershipState[recordBase + 5]$UDINT <> OwnerGeneration) |
			   (OwnershipState[recordBase + 6]$UDINT <>
			    CallerSessionEpoch) |
			   (OwnershipState[recordBase + 7]$UDINT <> RequestSequence) |
			   (OwnershipState[recordBase + 11]$UDINT <> expectedAxisMask) |
			   (OwnershipState[recordBase + 2] <> expectedOwnerKind) |
			   (OwnershipState[recordBase + 3] <> expectedCommandId) |
			   (OwnershipState[recordBase + 12] <> expectedReference) |
			   (OwnershipState[recordBase + 13] <>
			    expectedResourceKind) |
			   (OwnershipState[recordBase + 14] <>
			    expectedAdmissionMode) |
			   (OwnershipState[recordBase + 15]$UDINT <>
			    expectedIdentitySize) then
				Result := -2;
				RETURN;
			elsif OwnershipState[recordBase + 1] =
			      LMC_OWNER_STATE_QUARANTINED then
				Result := -3;
				RETURN;
			elsif OwnershipState[recordBase + 1] <>
			      LMC_OWNER_STATE_RESERVED then
				Result := -2;
				RETURN;
			end_if;
		elsif (OwnershipState[recordBase + 4]$UDINT = AdmissionToken) |
		      (OwnershipState[recordBase + 5]$UDINT = OwnerGeneration) then
			Result := -2;
			RETURN;
		end_if;
		axisIndex += 1;
	end_while;
	resourceValid := FALSE;
	case expectedResourceKind of
		LMC_OWNER_RESOURCE_AXIS:
			resourceValid :=
				(OwnershipState[7]$UDINT <> AdmissionToken) &
				(OwnershipState[8]$UDINT <> OwnerGeneration) &
				(OwnershipState[10]$UDINT <> AdmissionToken) &
				(OwnershipState[11]$UDINT <> OwnerGeneration) &
				(OwnershipState[13]$UDINT <> AdmissionToken) &
				(OwnershipState[14]$UDINT <> OwnerGeneration);
		LMC_OWNER_RESOURCE_LMC_HOME_ENGINE:
			resourceValid :=
				(OwnershipState[7]$UDINT = AdmissionToken) &
				(OwnershipState[8]$UDINT = OwnerGeneration) &
				(OwnershipState[9]$UDINT = expectedAxisMask) &
				(OwnershipState[10]$UDINT <> AdmissionToken) &
				(OwnershipState[11]$UDINT <> OwnerGeneration) &
				(OwnershipState[13]$UDINT <> AdmissionToken) &
				(OwnershipState[14]$UDINT <> OwnerGeneration);
		LMC_OWNER_RESOURCE_DS402_HOME_ENGINE:
			resourceValid :=
				(OwnershipState[10]$UDINT = AdmissionToken) &
				(OwnershipState[11]$UDINT = OwnerGeneration) &
				(OwnershipState[12]$UDINT = expectedAxisMask) &
				(OwnershipState[7]$UDINT <> AdmissionToken) &
				(OwnershipState[8]$UDINT <> OwnerGeneration) &
				(OwnershipState[13]$UDINT <> AdmissionToken) &
				(OwnershipState[14]$UDINT <> OwnerGeneration);
		LMC_OWNER_RESOURCE_DIAGNOSTICS_SDO_ENGINE:
			resourceValid :=
				(OwnershipState[13]$UDINT = AdmissionToken) &
				(OwnershipState[14]$UDINT = OwnerGeneration) &
				(OwnershipState[15]$UDINT = expectedAxisMask) &
				(OwnershipState[7]$UDINT <> AdmissionToken) &
				(OwnershipState[8]$UDINT <> OwnerGeneration) &
				(OwnershipState[10]$UDINT <> AdmissionToken) &
				(OwnershipState[11]$UDINT <> OwnerGeneration);
	else
	end_case;
	if resourceValid = FALSE then
		Result := -2;
		RETURN;
	end_if;

	// Choose an immutable exact bank before the first rollback mutation.
	if Reason = 0 then
		if OwnershipPreemptedIdentityState[
		   LMC_OWNER_PREEMPT_HEADER_BASE]$UDINT =
		   LMC_OWNER_PREEMPT_IDENTITY_MAGIC then
			preemptFlags := OwnershipPreemptedIdentityState[
				LMC_OWNER_PREEMPT_HEADER_BASE + 1]$UDINT;
			cleanupRequiredMask := OwnershipPreemptedIdentityState[
				LMC_OWNER_PREEMPT_HEADER_BASE + 8]$UDINT;
			cleanupCompleteMask := OwnershipPreemptedIdentityState[
				LMC_OWNER_PREEMPT_HEADER_BASE + 9]$UDINT;
			restorePreempt :=
				((preemptFlags and 0x0000FFFF) =
				 LMC_OWNER_IDENTITY_VERSION) &
				((preemptFlags and 0xFFFE0000) = 0) &
				(OwnershipPreemptedIdentityState[
				 LMC_OWNER_PREEMPT_HEADER_BASE + 2]$UDINT =
				 AdmissionToken) &
				(OwnershipPreemptedIdentityState[
				 LMC_OWNER_PREEMPT_HEADER_BASE + 3]$UDINT =
				 OwnerGeneration) &
				(OwnershipPreemptedIdentityState[
				 LMC_OWNER_PREEMPT_HEADER_BASE + 4]$UDINT =
				 expectedAxisMask) &
				(OwnershipPreemptedIdentityState[
				 LMC_OWNER_PREEMPT_HEADER_BASE + 5]$UDINT =
				 CallerSessionEpoch) &
				(OwnershipPreemptedIdentityState[
				 LMC_OWNER_PREEMPT_HEADER_BASE + 6]$UDINT =
				 RequestSequence) &
				(OwnershipPreemptedIdentityState[
				 LMC_OWNER_PREEMPT_HEADER_BASE + 7]$UDINT =
				 (TO_UDINT(expectedCommandId) or
				  (TO_UDINT(expectedReference) shl 16))) &
				((cleanupRequiredMask and (not expectedAxisMask)) = 0) &
				((cleanupCompleteMask and
				  (not cleanupRequiredMask)) = 0);
			if restorePreempt = FALSE then
				Result := -3;
				RETURN;
			end_if;
		else
			preemptBankValid := TRUE;
			identityIndex := 0;
			while identityIndex <= 323 do
				if OwnershipPreemptedState[identityIndex] <> 0 then
					preemptBankValid := FALSE;
				end_if;
				identityIndex += 1;
			end_while;
			identityIndex := 0;
			while identityIndex <= 431 do
				if OwnershipPreemptedIdentityState[identityIndex] <> 0 then
					preemptBankValid := FALSE;
				end_if;
				identityIndex += 1;
			end_while;
			if preemptBankValid = FALSE then
				Result := -3;
				RETURN;
			end_if;
		end_if;
		if restorePreempt = FALSE then
			restoreLease :=
				(expectedResourceKind = LMC_OWNER_RESOURCE_AXIS) &
				(expectedOwnerKind = LMC_OWNER_KIND_GROUP) &
				((expectedCommandId = 0x20A4) |
				 (expectedCommandId = 0x7D22) |
				 (expectedCommandId = 0x2048) |
				 (expectedCommandId = 0x2085)) &
				(OwnershipLeaseIdentityState[
				 LMC_OWNER_LEASE_IDENTITY_HEADER_BASE]$UDINT =
				 LMC_OWNER_LEASE_IDENTITY_MAGIC);
		end_if;
		if ((expectedCommandId = 0x20A4) |
		    (expectedCommandId = 0x7D22)) &
		   (restorePreempt = FALSE) & (restoreLease = FALSE) then
			Result := -3;
			RETURN;
		end_if;
	end_if;

	if restorePreempt | restoreLease then
		if restorePreempt then
			preemptBankValid := TRUE;
			restoredGroupActive := FALSE;
			restoredGroupFound := FALSE;
			restoredNonSafetyFound := FALSE;
			restoredGroupMask := 0;
			axisIndex := 1;
			while axisIndex <= LMC_OWNER_AXIS_COUNT do
				case axisIndex of
					1: axisBit := 0x00000001;
					2: axisBit := 0x00000002;
					3: axisBit := 0x00000004;
					4: axisBit := 0x00000008;
					5: axisBit := 0x00000010;
					6: axisBit := 0x00000020;
					7: axisBit := 0x00000040;
					8: axisBit := 0x00000080;
					9: axisBit := 0x00000100;
				else
					axisBit := 0;
				end_case;
				recordBase := (axisIndex - 1) * LMC_OWNER_AXIS_STRIDE;
				observerBase := (axisIndex - 1) * LMC_OWNER_OBSERVER_STRIDE;
				if (OwnershipPreemptedState[recordBase] <> axisIndex) |
				   (OwnershipPreemptedState[recordBase + 35]$UDINT <>
				    (LMC_OWNER_AXIS_RECORD_MAGIC + TO_UDINT(axisIndex))) then
					preemptBankValid := FALSE;
				end_if;
				snapshotState := OwnershipPreemptedState[recordBase + 1];
				snapshotOwnerKind := OwnershipPreemptedState[recordBase + 2];
				snapshotCommand := OwnershipPreemptedState[recordBase + 3];
				snapshotToken := OwnershipPreemptedState[recordBase + 4]$UDINT;
				snapshotGeneration :=
					OwnershipPreemptedState[recordBase + 5]$UDINT;
				snapshotSession := OwnershipPreemptedState[recordBase + 6]$UDINT;
				snapshotSequence := OwnershipPreemptedState[recordBase + 7]$UDINT;
				snapshotMask := OwnershipPreemptedState[recordBase + 11]$UDINT;
				snapshotReference := OwnershipPreemptedState[recordBase + 12];
				snapshotResourceKind := OwnershipPreemptedState[recordBase + 13];
				snapshotAdmissionMode := OwnershipPreemptedState[recordBase + 14];
				snapshotIdentitySize :=
					OwnershipPreemptedState[recordBase + 15]$UDINT;
				observersIdle := TRUE;
				observerIndex := 0;
				while observerIndex < LMC_OWNER_OBSERVER_STRIDE do
					if OwnershipPreemptedIdentityState[
					   LMC_OWNER_PREEMPT_OBSERVER_BASE + observerBase +
					   observerIndex] <> 0 then
						observersIdle := FALSE;
					end_if;
					observerIndex += 1;
				end_while;
				if snapshotState = LMC_OWNER_STATE_IDLE then
					if (snapshotOwnerKind <> 0) | (snapshotCommand <> 0) |
					   (snapshotToken <> 0) | (snapshotGeneration <> 0) |
					   (snapshotSession <> 0) | (snapshotSequence <> 0) |
					   (snapshotMask <> 0) | (snapshotReference <> 0) |
					   (snapshotResourceKind <> 0) |
					   (snapshotAdmissionMode <> 0) |
					   (snapshotIdentitySize <> 0) |
					   (observersIdle = FALSE) then
						preemptBankValid := FALSE;
					end_if;
				else
					identityExpectedSize := 0;
					if snapshotCommand = 0x2023 then
						identityExpectedSize := 8;
					elsif snapshotCommand = 0x2024 then
						identityExpectedSize := 1;
					elsif snapshotCommand = 0x2022 then
						identityExpectedSize := 16;
					elsif (snapshotCommand = 0x209F) |
					      (snapshotCommand = 0x20A0) then
						identityExpectedSize := 32;
					elsif snapshotCommand = 0x20A2 then
						identityExpectedSize := 24;
					elsif (snapshotCommand = 0x2047) |
					      (snapshotCommand = 0x2048) |
					      (snapshotCommand = 0x2049) |
					      (snapshotCommand = 0x204A) |
					      (snapshotCommand = 0x204B) then
						identityExpectedSize := 1;
					elsif snapshotCommand = 0x2085 then
						identityExpectedSize := 16;
					elsif snapshotCommand = 0x20A4 then
						identityExpectedSize := 96;
					elsif snapshotCommand = 0x7D22 then
						identityExpectedSize := 104;
					elsif snapshotCommand = 0x20E7 then
						identityExpectedSize := 1320;
					elsif snapshotCommand = 0x7D13 then
						identityExpectedSize := 56;
					elsif (snapshotCommand = 0x7D15) |
					      (snapshotCommand = 0x7E53) then
						identityExpectedSize := 72;
					end_if;
					probeAxisBit := 0;
					case snapshotReference of
						1: probeAxisBit := 0x00000001;
						2: probeAxisBit := 0x00000002;
						3: probeAxisBit := 0x00000004;
						4: probeAxisBit := 0x00000008;
						5: probeAxisBit := 0x00000010;
						6: probeAxisBit := 0x00000020;
						7: probeAxisBit := 0x00000040;
						8: probeAxisBit := 0x00000080;
						9: probeAxisBit := 0x00000100;
					else
					end_case;
					snapshotTupleValid := FALSE;
					case snapshotOwnerKind of
						LMC_OWNER_KIND_DIRECT:
							snapshotTupleValid :=
								(snapshotResourceKind =
								 LMC_OWNER_RESOURCE_AXIS) &
								(probeAxisBit <> 0) &
								((snapshotMask and probeAxisBit) <> 0) &
								((snapshotState = LMC_OWNER_STATE_RESERVED) |
								 (snapshotState =
								  LMC_OWNER_STATE_DIRECT_ACTIVE) |
								 (snapshotState =
								  LMC_OWNER_STATE_QUARANTINED));
							if snapshotCommand = 0x2022 then
								snapshotTupleValid := snapshotTupleValid &
									(snapshotAdmissionMode =
									 LMC_OWNER_ADMISSION_SAFETY);
							elsif snapshotCommand = 0x2023 then
								snapshotTupleValid := snapshotTupleValid &
									((snapshotAdmissionMode =
									  LMC_OWNER_ADMISSION_ORDINARY) |
									 (snapshotAdmissionMode =
									  LMC_OWNER_ADMISSION_SAFETY));
							elsif (snapshotCommand = 0x2024) |
							      (snapshotCommand = 0x209F) |
							      (snapshotCommand = 0x20A0) |
							      (snapshotCommand = 0x20A2) then
								snapshotTupleValid := snapshotTupleValid &
									(snapshotAdmissionMode =
									 LMC_OWNER_ADMISSION_ORDINARY);
							else
								snapshotTupleValid := FALSE;
							end_if;
						LMC_OWNER_KIND_GROUP:
							snapshotTupleValid :=
								(snapshotResourceKind =
								 LMC_OWNER_RESOURCE_AXIS) &
								(snapshotReference = 0x0100) &
								((snapshotState = LMC_OWNER_STATE_RESERVED) |
								 (snapshotState = LMC_OWNER_STATE_GROUP_LEASE) |
								 (snapshotState = LMC_OWNER_STATE_GROUP_ACTIVE) |
								 (snapshotState =
								  LMC_OWNER_STATE_QUARANTINED));
							if (snapshotCommand = 0x2047) |
							   (snapshotCommand = 0x20A4) |
							   (snapshotCommand = 0x7D22) then
								snapshotTupleValid := snapshotTupleValid &
									(snapshotAdmissionMode =
									 LMC_OWNER_ADMISSION_ORDINARY) &
									(snapshotMask =
									 LMC_OWNER_PROFILE_AXIS_MASK);
							elsif snapshotCommand = 0x2048 then
								snapshotTupleValid := snapshotTupleValid &
									(snapshotAdmissionMode =
									 LMC_OWNER_ADMISSION_SAFETY) &
									(snapshotMask =
									 LMC_OWNER_PROFILE_AXIS_MASK);
							elsif snapshotCommand = 0x2085 then
								snapshotTupleValid := snapshotTupleValid &
									(snapshotAdmissionMode =
									 LMC_OWNER_ADMISSION_SAFETY) &
									((snapshotMask =
									  LMC_OWNER_PROFILE_AXIS_MASK) |
									 (snapshotMask =
									  LMC_OWNER_ROBOT_AXIS_MASK));
							elsif (snapshotCommand = 0x2049) |
							      (snapshotCommand = 0x204A) then
								snapshotTupleValid := snapshotTupleValid &
									(snapshotAdmissionMode =
									 LMC_OWNER_ADMISSION_ORDINARY) &
									(snapshotMask =
									 LMC_OWNER_ROBOT_AXIS_MASK);
							elsif snapshotCommand = 0x204B then
								snapshotTupleValid := snapshotTupleValid &
									(snapshotAdmissionMode =
									 LMC_OWNER_ADMISSION_SAFETY) &
									(snapshotMask =
									 LMC_OWNER_ROBOT_AXIS_MASK);
							elsif snapshotCommand = 0x20E7 then
								snapshotTupleValid := snapshotTupleValid &
									(snapshotAdmissionMode =
									 LMC_OWNER_ADMISSION_LIFECYCLE) &
									(snapshotMask =
									 LMC_OWNER_ROBOT_AXIS_MASK);
							else
								snapshotTupleValid := FALSE;
							end_if;
						LMC_OWNER_KIND_LMC_HOME:
							snapshotTupleValid :=
								(snapshotCommand = 0x7D13) &
								(snapshotResourceKind =
								 LMC_OWNER_RESOURCE_LMC_HOME_ENGINE) &
								(snapshotAdmissionMode =
								 LMC_OWNER_ADMISSION_LIFECYCLE) &
								(probeAxisBit <> 0) &
								(probeAxisBit <= 0x00000008) &
								(snapshotMask = probeAxisBit) &
								((snapshotState = LMC_OWNER_STATE_RESERVED) |
								 (snapshotState =
								  LMC_OWNER_STATE_LMC_HOME_ACTIVE) |
								 (snapshotState =
								  LMC_OWNER_STATE_QUARANTINED));
						LMC_OWNER_KIND_DS402_HOME:
							snapshotTupleValid :=
								(snapshotCommand = 0x7D15) &
								(snapshotResourceKind =
								 LMC_OWNER_RESOURCE_DS402_HOME_ENGINE) &
								(snapshotAdmissionMode =
								 LMC_OWNER_ADMISSION_LIFECYCLE) &
								(probeAxisBit <> 0) &
								(probeAxisBit <= 0x00000008) &
								(snapshotMask = probeAxisBit) &
								((snapshotState = LMC_OWNER_STATE_RESERVED) |
								 (snapshotState =
								  LMC_OWNER_STATE_DS402_HOME_ACTIVE) |
								 (snapshotState =
								  LMC_OWNER_STATE_QUARANTINED));
						LMC_OWNER_KIND_ENCODER:
							snapshotTupleValid :=
								(snapshotCommand = 0x7E53) &
								(snapshotResourceKind =
								 LMC_OWNER_RESOURCE_DIAGNOSTICS_SDO_ENGINE) &
								(snapshotAdmissionMode =
								 LMC_OWNER_ADMISSION_LIFECYCLE) &
								(probeAxisBit <> 0) &
								(probeAxisBit <= 0x00000008) &
								(snapshotMask = probeAxisBit) &
								((snapshotState = LMC_OWNER_STATE_RESERVED) |
								 (snapshotState =
								  LMC_OWNER_STATE_TW20_QUEUED) |
								 (snapshotState =
								  LMC_OWNER_STATE_TW20_RUNNING) |
								 (snapshotState =
								  LMC_OWNER_STATE_TW20_DRAINING) |
								 (snapshotState =
								  LMC_OWNER_STATE_QUARANTINED));
					else
					end_case;
					identityShapeValid :=
						(identityExpectedSize <> 0) &
						(snapshotIdentitySize = identityExpectedSize) &
						(snapshotToken <> 0) & (snapshotGeneration <> 0) &
						(snapshotSession <> 0) & (snapshotSequence <> 0) &
						(snapshotMask <> 0) &
						(snapshotMask <= LMC_OWNER_ROBOT_AXIS_MASK) &
						((snapshotMask and axisBit) <> 0);
					identityPrefixSize := snapshotIdentitySize;
					if identityPrefixSize >
					   LMC_OWNER_IDENTITY_PREFIX_BYTES then
						identityPrefixSize := LMC_OWNER_IDENTITY_PREFIX_BYTES;
					end_if;
					identityTailSize := 0;
					if snapshotIdentitySize >
					   LMC_OWNER_IDENTITY_PREFIX_BYTES then
						identityTailSize := snapshotIdentitySize -
							LMC_OWNER_IDENTITY_PREFIX_BYTES;
					end_if;
					identityTailOffset := 0;
					if snapshotOwnerKind <> LMC_OWNER_KIND_GROUP then
						if (snapshotReference < 1) |
						   (snapshotReference > LMC_OWNER_AXIS_COUNT) |
						   (identityTailSize > 8) then
							identityShapeValid := FALSE;
						else
							identityTailOffset :=
								TO_UDINT(snapshotReference - 1) * 8;
						end_if;
					end_if;
					if (identityTailOffset + identityTailSize) >
					   LMC_OWNER_IDENTITY_SUFFIX_BYTES then
						identityShapeValid := FALSE;
					end_if;
					if (snapshotTupleValid = FALSE) |
					   (identityShapeValid = FALSE) then
						preemptBankValid := FALSE;
					end_if;
					if (snapshotOwnerKind <> LMC_OWNER_KIND_GROUP) &
					   (snapshotAdmissionMode <>
					    LMC_OWNER_ADMISSION_SAFETY) then
						restoredNonSafetyFound := TRUE;
					end_if;
					// The live compact identity table has one Group header. Therefore
					// every non-idle Group snapshot must be one globally coherent
					// tuple before any selected member can be restored.
					if snapshotOwnerKind = LMC_OWNER_KIND_GROUP then
						if restoredGroupFound = FALSE then
							restoredGroupFound := TRUE;
							restoredGroupToken := snapshotToken;
							restoredGroupGeneration := snapshotGeneration;
							restoredGroupSession := snapshotSession;
							restoredGroupSequence := snapshotSequence;
							restoredGroupMask := snapshotMask;
							restoredGroupCommand := snapshotCommand;
							restoredGroupReference := snapshotReference;
							restoredGroupState := snapshotState;
							restoredGroupAdmissionMode :=
								snapshotAdmissionMode;
							restoredGroupIdentitySize := snapshotIdentitySize;
						elsif (restoredGroupToken <> snapshotToken) |
						      (restoredGroupGeneration <> snapshotGeneration) |
						      (restoredGroupSession <> snapshotSession) |
						      (restoredGroupSequence <> snapshotSequence) |
						      (restoredGroupMask <> snapshotMask) |
						      (restoredGroupCommand <> snapshotCommand) |
						      (restoredGroupReference <> snapshotReference) |
						      (restoredGroupState <> snapshotState) |
						      (restoredGroupAdmissionMode <>
						       snapshotAdmissionMode) |
						      (restoredGroupIdentitySize <>
						       snapshotIdentitySize) then
							preemptBankValid := FALSE;
						end_if;
					end_if;
					probeAxisIndex := 1;
					while probeAxisIndex <= LMC_OWNER_AXIS_COUNT do
						case probeAxisIndex of
							1: probeAxisBit := 0x00000001;
							2: probeAxisBit := 0x00000002;
							3: probeAxisBit := 0x00000004;
							4: probeAxisBit := 0x00000008;
							5: probeAxisBit := 0x00000010;
							6: probeAxisBit := 0x00000020;
							7: probeAxisBit := 0x00000040;
							8: probeAxisBit := 0x00000080;
							9: probeAxisBit := 0x00000100;
						else
							probeAxisBit := 0;
						end_case;
						probeRecordBase := (probeAxisIndex - 1) *
							LMC_OWNER_AXIS_STRIDE;
						if (snapshotMask and probeAxisBit) <> 0 then
							if (OwnershipPreemptedState[
							    probeRecordBase + 1] <> snapshotState) |
							   (OwnershipPreemptedState[
							    probeRecordBase + 2] <> snapshotOwnerKind) |
							   (OwnershipPreemptedState[
							    probeRecordBase + 3] <> snapshotCommand) |
							   (OwnershipPreemptedState[
							    probeRecordBase + 4]$UDINT <> snapshotToken) |
							   (OwnershipPreemptedState[
							    probeRecordBase + 5]$UDINT <>
							    snapshotGeneration) |
							   (OwnershipPreemptedState[
							    probeRecordBase + 6]$UDINT <> snapshotSession) |
							   (OwnershipPreemptedState[
							    probeRecordBase + 7]$UDINT <> snapshotSequence) |
							   (OwnershipPreemptedState[
							    probeRecordBase + 11]$UDINT <> snapshotMask) |
							   (OwnershipPreemptedState[
							    probeRecordBase + 12] <> snapshotReference) |
							   (OwnershipPreemptedState[
							    probeRecordBase + 13] <>
							    snapshotResourceKind) |
							   (OwnershipPreemptedState[
							    probeRecordBase + 14] <>
							    snapshotAdmissionMode) |
							   (OwnershipPreemptedState[
							    probeRecordBase + 15]$UDINT <>
							    snapshotIdentitySize) then
								preemptBankValid := FALSE;
							end_if;
							identityCompareResult := _memcmp(
								ptr1:=#OwnershipPreemptedState[
								 recordBase + 16],
								ptr2:=#OwnershipPreemptedState[
								 probeRecordBase + 16],
								cntr:=identityPrefixSize);
							if identityCompareResult <> 0 then
								preemptBankValid := FALSE;
							end_if;
						elsif (OwnershipPreemptedState[
						       probeRecordBase + 4]$UDINT = snapshotToken) |
						      (OwnershipPreemptedState[
						       probeRecordBase + 5]$UDINT =
						       snapshotGeneration) then
							preemptBankValid := FALSE;
						end_if;
						probeAxisIndex += 1;
					end_while;
					observerSnapshotValid := observersIdle &
						(snapshotState = LMC_OWNER_STATE_GROUP_LEASE);
					if observersIdle = FALSE then
						observerSnapshotValid :=
							(OwnershipPreemptedIdentityState[
							 LMC_OWNER_PREEMPT_OBSERVER_BASE +
							 observerBase]$UDINT =
							 (LMC_OWNER_OBSERVER_MAGIC + TO_UDINT(axisIndex))) &
							((OwnershipPreemptedIdentityState[
							  LMC_OWNER_PREEMPT_OBSERVER_BASE +
							  observerBase + 5]$UDINT and
							  (0xFFFFFFFF xor LMC_OWNER_OBSERVER_KNOWN_MASK)) = 0) &
							(((OwnershipPreemptedIdentityState[
							   LMC_OWNER_PREEMPT_OBSERVER_BASE +
							   observerBase + 1]$UDINT = 0) &
							  (OwnershipPreemptedIdentityState[
							   LMC_OWNER_PREEMPT_OBSERVER_BASE +
							   observerBase + 2]$UDINT = 0)) |
							 ((OwnershipPreemptedIdentityState[
							   LMC_OWNER_PREEMPT_OBSERVER_BASE +
							   observerBase + 1]$UDINT = snapshotToken) &
							  (OwnershipPreemptedIdentityState[
							   LMC_OWNER_PREEMPT_OBSERVER_BASE +
							   observerBase + 2]$UDINT =
							   snapshotGeneration)));
					end_if;
					if observerSnapshotValid = FALSE then
						preemptBankValid := FALSE;
					end_if;
					if (snapshotState = LMC_OWNER_STATE_GROUP_ACTIVE) &
					   (snapshotOwnerKind = LMC_OWNER_KIND_GROUP) then
						restoredGroupActive := TRUE;
						// A disjoint Group owner remains live during this rollback.
						// Prove its complete live tuple/header/observer against the
						// exact all-axis snapshot before retaining the lease bank.
						if (expectedAxisMask and axisBit) = 0 then
							probeRecordBase := LMC_OWNER_GLOBAL_SLOTS + recordBase;
							if (OwnershipState[probeRecordBase] <> axisIndex) |
							   (OwnershipState[probeRecordBase + 35]$UDINT <>
							    (LMC_OWNER_AXIS_RECORD_MAGIC + TO_UDINT(axisIndex))) |
							   (OwnershipState[probeRecordBase + 1] <> snapshotState) |
							   (OwnershipState[probeRecordBase + 2] <>
							    snapshotOwnerKind) |
							   (OwnershipState[probeRecordBase + 3] <> snapshotCommand) |
							   (OwnershipState[probeRecordBase + 4]$UDINT <>
							    snapshotToken) |
							   (OwnershipState[probeRecordBase + 5]$UDINT <>
							    snapshotGeneration) |
							   (OwnershipState[probeRecordBase + 6]$UDINT <>
							    snapshotSession) |
							   (OwnershipState[probeRecordBase + 7]$UDINT <>
							    snapshotSequence) |
							   (OwnershipState[probeRecordBase + 11]$UDINT <>
							    snapshotMask) |
							   (OwnershipState[probeRecordBase + 12] <>
							    snapshotReference) |
							   (OwnershipState[probeRecordBase + 13] <>
							    snapshotResourceKind) |
							   (OwnershipState[probeRecordBase + 14] <>
							    snapshotAdmissionMode) |
							   (OwnershipState[probeRecordBase + 15]$UDINT <>
							    snapshotIdentitySize) then
								preemptBankValid := FALSE;
							end_if;
							identityCompareResult := _memcmp(
								ptr1:=#OwnershipState[probeRecordBase + 16],
								ptr2:=#OwnershipPreemptedState[recordBase + 16],
								cntr:=identityPrefixSize);
							if identityCompareResult <> 0 then
								preemptBankValid := FALSE;
							end_if;
							identityCompareResult := _memcmp(
								ptr1:=#OwnershipObserverState[observerBase],
								ptr2:=#OwnershipPreemptedIdentityState[
								 LMC_OWNER_PREEMPT_OBSERVER_BASE + observerBase],
								cntr:=LMC_OWNER_OBSERVER_STRIDE * 4);
							if identityCompareResult <> 0 then
								preemptBankValid := FALSE;
							end_if;
							identityHeaderBase :=
								LMC_OWNER_IDENTITY_GROUP_HEADER_BASE;
							if (OwnershipIdentityState[identityHeaderBase]$UDINT <>
							    LMC_OWNER_IDENTITY_GROUP_MAGIC) |
							   (OwnershipIdentityState[identityHeaderBase + 1] <>
							    LMC_OWNER_IDENTITY_VERSION) |
							   (OwnershipIdentityState[identityHeaderBase + 2]$UDINT <>
							    snapshotIdentitySize) |
							   (OwnershipIdentityState[identityHeaderBase + 3]$UDINT <>
							    snapshotToken) |
							   (OwnershipIdentityState[identityHeaderBase + 4]$UDINT <>
							    snapshotGeneration) |
							   (OwnershipIdentityState[identityHeaderBase + 5]$UDINT <>
							    snapshotMask) |
							   (OwnershipIdentityState[identityHeaderBase + 6]$UDINT <>
							    snapshotSession) |
							   (OwnershipIdentityState[identityHeaderBase + 7]$UDINT <>
							    snapshotSequence) |
							   (OwnershipIdentityState[identityHeaderBase + 8]$UDINT <>
							    (TO_UDINT(snapshotCommand) or
							     (TO_UDINT(snapshotReference) shl 16))) |
							   (OwnershipIdentityState[identityHeaderBase + 9]$UDINT <>
							    (TO_UDINT(snapshotOwnerKind) or
							     (TO_UDINT(snapshotResourceKind) shl 8) or
							     (TO_UDINT(snapshotAdmissionMode) shl 16))) then
								preemptBankValid := FALSE;
							end_if;
						end_if;
					end_if;
				end_if;
				axisIndex += 1;
			end_while;
			if restoredGroupFound & restoredNonSafetyFound then
				preemptBankValid := FALSE;
			end_if;
			if preemptBankValid = FALSE then
				Result := -3;
				RETURN;
			end_if;
		end_if;
		// A restored active Group record requires its exact underlying 0x2047
		// lease to remain available. A direct lease restore consumes the same
		// bank. Validate the complete lease before changing any live record.
		if restoreLease | restoredGroupActive then
			leaseExpectedMask := expectedAxisMask;
			if restoredGroupActive then
				leaseExpectedMask := restoredGroupMask;
			end_if;
			leaseBankValid :=
				(leaseExpectedMask = LMC_OWNER_PROFILE_AXIS_MASK) &
				(OwnershipLeaseIdentityState[
				 LMC_OWNER_LEASE_IDENTITY_HEADER_BASE]$UDINT =
				 LMC_OWNER_LEASE_IDENTITY_MAGIC) &
				(OwnershipLeaseIdentityState[
				 LMC_OWNER_LEASE_IDENTITY_HEADER_BASE + 1] =
				 LMC_OWNER_IDENTITY_VERSION) &
				(OwnershipLeaseIdentityState[
				 LMC_OWNER_LEASE_IDENTITY_HEADER_BASE + 2]$UDINT = 1) &
				(OwnershipLeaseIdentityState[
				 LMC_OWNER_LEASE_IDENTITY_HEADER_BASE + 3]$UDINT <> 0) &
				(OwnershipLeaseIdentityState[
				 LMC_OWNER_LEASE_IDENTITY_HEADER_BASE + 4]$UDINT <> 0) &
				(OwnershipLeaseIdentityState[
				 LMC_OWNER_LEASE_IDENTITY_HEADER_BASE + 5]$UDINT =
				 leaseExpectedMask) &
				(OwnershipLeaseIdentityState[
				 LMC_OWNER_LEASE_IDENTITY_HEADER_BASE + 6]$UDINT <> 0) &
				(OwnershipLeaseIdentityState[
				 LMC_OWNER_LEASE_IDENTITY_HEADER_BASE + 7]$UDINT <> 0) &
				(OwnershipLeaseIdentityState[
				 LMC_OWNER_LEASE_IDENTITY_HEADER_BASE + 8]$UDINT =
				 (TO_UDINT(0x2047) or (TO_UDINT(0x0100) shl 16))) &
				(OwnershipLeaseIdentityState[
				 LMC_OWNER_LEASE_IDENTITY_HEADER_BASE + 9]$UDINT =
				 (TO_UDINT(LMC_OWNER_KIND_GROUP) or
				  (TO_UDINT(LMC_OWNER_RESOURCE_AXIS) shl 8) or
				  (TO_UDINT(LMC_OWNER_ADMISSION_ORDINARY) shl 16)));
			firstRecordBase := -1;
			axisIndex := 1;
			while axisIndex <= LMC_OWNER_AXIS_COUNT do
				case axisIndex of
					1: axisBit := 0x00000001;
					2: axisBit := 0x00000002;
					3: axisBit := 0x00000004;
					4: axisBit := 0x00000008;
					5: axisBit := 0x00000010;
					6: axisBit := 0x00000020;
					7: axisBit := 0x00000040;
					8: axisBit := 0x00000080;
					9: axisBit := 0x00000100;
				else
					axisBit := 0;
				end_case;
				recordBase := (axisIndex - 1) * LMC_OWNER_AXIS_STRIDE;
				if (OwnershipLeaseState[recordBase] <> axisIndex) |
				   (OwnershipLeaseState[recordBase + 35]$UDINT <>
				    (LMC_OWNER_AXIS_RECORD_MAGIC + TO_UDINT(axisIndex))) then
					leaseBankValid := FALSE;
				end_if;
				if (leaseExpectedMask and axisBit) <> 0 then
					if (OwnershipLeaseState[recordBase + 1] <>
					    LMC_OWNER_STATE_GROUP_LEASE) |
					   (OwnershipLeaseState[recordBase + 2] <>
					    LMC_OWNER_KIND_GROUP) |
					   (OwnershipLeaseState[recordBase + 3] <> 0x2047) |
					   (OwnershipLeaseState[recordBase + 4]$UDINT <>
					    OwnershipLeaseIdentityState[
					     LMC_OWNER_LEASE_IDENTITY_HEADER_BASE + 3]$UDINT) |
					   (OwnershipLeaseState[recordBase + 5]$UDINT <>
					    OwnershipLeaseIdentityState[
					     LMC_OWNER_LEASE_IDENTITY_HEADER_BASE + 4]$UDINT) |
					   (OwnershipLeaseState[recordBase + 6]$UDINT <>
					    OwnershipLeaseIdentityState[
					     LMC_OWNER_LEASE_IDENTITY_HEADER_BASE + 6]$UDINT) |
					   (OwnershipLeaseState[recordBase + 7]$UDINT <>
					    OwnershipLeaseIdentityState[
					     LMC_OWNER_LEASE_IDENTITY_HEADER_BASE + 7]$UDINT) |
					   (OwnershipLeaseState[recordBase + 11]$UDINT <>
					    leaseExpectedMask) |
					   (OwnershipLeaseState[recordBase + 12] <> 0x0100) |
					   (OwnershipLeaseState[recordBase + 13] <>
					    LMC_OWNER_RESOURCE_AXIS) |
					   (OwnershipLeaseState[recordBase + 14] <>
					    LMC_OWNER_ADMISSION_ORDINARY) |
					   (OwnershipLeaseState[recordBase + 15]$UDINT <> 1) |
					   (OwnershipLeaseState[recordBase + 16]$UDINT <> 1) then
						leaseBankValid := FALSE;
					end_if;
					identityIndex := 17;
					while identityIndex <= 31 do
						if OwnershipLeaseState[recordBase + identityIndex] <> 0 then
							leaseBankValid := FALSE;
						end_if;
						identityIndex += 1;
					end_while;
					if firstRecordBase < 0 then
						firstRecordBase := recordBase;
					else
						identityCompareResult := _memcmp(
							ptr1:=#OwnershipLeaseState[firstRecordBase + 16],
							ptr2:=#OwnershipLeaseState[recordBase + 16], cntr:=1);
						if identityCompareResult <> 0 then
							leaseBankValid := FALSE;
						end_if;
					end_if;
				else
					if (OwnershipLeaseState[recordBase + 4]$UDINT =
					    OwnershipLeaseIdentityState[
					     LMC_OWNER_LEASE_IDENTITY_HEADER_BASE + 3]$UDINT) |
					   (OwnershipLeaseState[recordBase + 5]$UDINT =
					    OwnershipLeaseIdentityState[
					     LMC_OWNER_LEASE_IDENTITY_HEADER_BASE + 4]$UDINT) then
						leaseBankValid := FALSE;
					end_if;
					identityIndex := 1;
					while identityIndex <= 34 do
						if OwnershipLeaseState[recordBase + identityIndex] <> 0 then
							leaseBankValid := FALSE;
						end_if;
						identityIndex += 1;
					end_while;
				end_if;
				axisIndex += 1;
			end_while;
			identityIndex := 0;
			while identityIndex < LMC_OWNER_IDENTITY_SUFFIX_DINTS do
				if OwnershipLeaseIdentityState[identityIndex] <> 0 then
					leaseBankValid := FALSE;
				end_if;
				identityIndex += 1;
			end_while;
			if (leaseBankValid = FALSE) | (firstRecordBase < 0) then
				OwnershipState[24] := 1;
				Result := -3;
				RETURN;
			end_if;
		end_if;
